LIN {X 0,Y 474.316,Z 460.054,A -85,B 0,C 180,E1 -7102.337,E2 -7102.337} C_VEL
LIN {X 0,Y 474.18,Z 465.59,A -85,B 0,C 180,E1 -7103.233,E2 -7103.233} C_VEL
LIN {X 0,Y 474.066,Z 469.783,A -85,B 0,C 180,E1 -7104.044,E2 -7104.044} C_VEL
LIN {X 0,Y 473.822,Z 474.988,A -85,B 0,C 180,E1 -7105.321,E2 -7105.321} C_VEL
LIN {X 0,Y 473.855,Z 477.663,A -85,B 0,C 180,E1 -7106.173,E2 -7106.173} C_VEL
LIN {X 0,Y 473.746,Z 480.593,A -85,B 0,C 180,E1 -7107.449,E2 -7107.449} C_VEL
LIN {X 0,Y 473.697,Z 481.876,A -85,B 0,C 180,E1 -7108.3,E2 -7108.3} C_VEL
LIN {X 0,Y 473.685,Z 482.688,A -85,B 0,C 180,E1 -7109.15,E2 -7109.15} C_VEL
LIN {X 0,Y 473.668,Z 482.997,A -85,B 0,C 180,E1 -7110,E2 -7110} C_VEL
LIN {X 0,Y 473.686,Z 482.723,A -85,B 0,C 180,E1 -7110.85,E2 -7110.85} C_VEL
LIN {X 0,Y 473.695,Z 481.979,A -85,B 0,C 180,E1 -7111.7,E2 -7111.7} C_VEL
LIN {X 0,Y 473.728,Z 480.766,A -85,B 0,C 180,E1 -7112.551,E2 -7112.551} C_VEL
LIN {X 0,Y 473.852,Z 477.91,A -85,B 0,C 180,E1 -7113.827,E2 -7113.827} C_VEL
LIN {X 0,Y 473.817,Z 475.311,A -85,B 0,C 180,E1 -7114.679,E2 -7114.679} C_VEL
LIN {X 0,Y 474.052,Z 470.192,A -85,B 0,C 180,E1 -7115.957,E2 -7115.957} C_VEL
LIN {X 0,Y 474.188,Z 464.687,A -85,B 0,C 180,E1 -7117.023,E2 -7117.023} C_VEL
LIN {X 0,Y 474.404,Z 457.777,A -85,B 0,C 180,E1 -7118.09,E2 -7118.09} C_VEL
LIN {X 0,Y 474.692,Z 449.845,A -85,B 0,C 180,E1 -7119.05,E2 -7119.05} C_VEL
LIN {X 0,Y 474.987,Z 442.281,A -85,B 0,C 180,E1 -7119.797,E2 -7119.797} C_VEL
LIN {X 0,Y 475.274,Z 434.358,A -85,B 0,C 180,E1 -7120.436,E2 -7120.436} C_VEL
LIN {X 0,Y 475.551,Z 426.183,A -85,B 0,C 180,E1 -7120.969,E2 -7120.969} C_VEL
LIN {X 0,Y 475.774,Z 417.91,A -85,B 0,C 180,E1 -7121.395,E2 -7121.395} C_VEL
LIN {X 0,Y 475.954,Z 408.99,A -85,B 0,C 180,E1 -7121.741,E2 -7121.741} C_VEL
LIN {X 0,Y 476.163,Z 399.664,A -85,B 0,C 180,E1 -7121.987,E2 -7121.987} C_VEL
LIN {X 0,Y 476.373,Z 336.635,A -85,B 0,C 180,E1 -7122.957,E2 -7122.957} C_VEL
LIN {X 0,Y 474.583,Z 324.02,A -85,B 0,C 180,E1 -7123.223,E2 -7123.223} C_VEL
LIN {X 0,Y 474.544,Z 323.281,A -85,B 0,C 180,E1 -7123.314,E2 -7123.314} C_VEL
LIN {X 0,Y 474.924,Z 309.716,A -85,B 0,C 180,E1 -7126.329,E2 -7126.329} C_VEL
LIN {X 0,Y 475.429,Z 296.05,A -85,B 0,C 180,E1 -7129.426,E2 -7129.426} C_VEL
LIN {X 0,Y 475.34,Z 290.192,A -85,B 0,C 180,E1 -7130.783,E2 -7130.783} C_VEL
LIN {X 0,Y 474.664,Z 286.26,A -85,B 0,C 180,E1 -7131.782,E2 -7131.782} C_VEL
LIN {X 0,Y 474.625,Z 286.175,A -85,B 0,C 180,E1 -7134.494,E2 -7134.494} C_VEL
LIN {X 0,Y 474.598,Z 286.18,A -85,B 0,C 180,E1 -7137.326,E2 -7137.326} C_VEL
LIN {X 0,Y 474.594,Z 286.176,A -85,B 0,C 180,E1 -7140.23,E2 -7140.23} C_VEL
LIN {X 0,Y 474.612,Z 286.178,A -85,B 0,C 180,E1 -7143.222,E2 -7143.222} C_VEL
LIN {X 0,Y 474.58,Z 286.177,A -85,B 0,C 180,E1 -7146.323,E2 -7146.323} C_VEL
LIN {X 0,Y 474.618,Z 286.177,A -85,B 0,C 180,E1 -7149.547,E2 -7149.547} C_VEL
LIN {X 0,Y 474.571,Z 286.178,A -85,B 0,C 180,E1 -7152.229,E2 -7152.229} C_VEL
LIN {X 0,Y 474.61,Z 286.18,A -85,B 0,C 180,E1 -7155.297,E2 -7155.297} C_VEL
LIN {X 0,Y 474.585,Z 286.177,A -85,B 0,C 180,E1 -7158.211,E2 -7158.211} C_VEL
LIN {X 0,Y 474.601,Z 286.176,A -85,B 0,C 180,E1 -7161.541,E2 -7161.541} C_VEL
LIN {X 0,Y 474.611,Z 286.179,A -85,B 0,C 180,E1 -7164.724,E2 -7164.724} C_VEL
LIN {X 0,Y 474.617,Z 286.173,A -85,B 0,C 180,E1 -7167.786,E2 -7167.786} C_VEL
LIN {X 0,Y 474.589,Z 286.182,A -85,B 0,C 180,E1 -7170.89,E2 -7170.89} C_VEL
LIN {X 0,Y 474.58,Z 286.177,A -85,B 0,C 180,E1 -7173.623,E2 -7173.623} C_VEL
LIN {X 0,Y 474.624,Z 286.18,A -85,B 0,C 180,E1 -7176.642,E2 -7176.642} C_VEL
LIN {X 0,Y 474.631,Z 286.173,A -85,B 0,C 180,E1 -7180.088,E2 -7180.088} C_VEL
LIN {X 0,Y 474.578,Z 286.181,A -85,B 0,C 180,E1 -7182.772,E2 -7182.772} C_VEL
LIN {X 0,Y 474.621,Z 286.172,A -85,B 0,C 180,E1 -7185.42,E2 -7185.42} C_VEL
LIN {X 0,Y 474.693,Z 286.167,A -85,B 0,C 180,E1 -7188.037,E2 -7188.037} C_VEL
LIN {X 0,Y 474.696,Z 286.163,A -85,B 0,C 180,E1 -7191.486,E2 -7191.486} C_VEL
LIN {X 0,Y 474.728,Z 286.165,A -85,B 0,C 180,E1 -7194.052,E2 -7194.052} C_VEL
LIN {X 0,Y 474.86,Z 286.143,A -85,B 0,C 180,E1 -7197.455,E2 -7197.455} C_VEL
LIN {X 0,Y 474.868,Z 286.149,A -85,B 0,C 180,E1 -7200,E2 -7200} C_VEL
LIN {X 0,Y 474.859,Z 286.144,A -85,B 0,C 180,E1 -7202.545,E2 -7202.545} C_VEL
LIN {X 0,Y 474.726,Z 286.166,A -85,B 0,C 180,E1 -7205.948,E2 -7205.948} C_VEL
LIN {X 0,Y 474.652,Z 286.169,A -85,B 0,C 180,E1 -7208.515,E2 -7208.515} C_VEL
LIN {X 0,Y 474.681,Z 286.169,A -85,B 0,C 180,E1 -7211.963,E2 -7211.963} C_VEL
LIN {X 0,Y 474.676,Z 286.171,A -85,B 0,C 180,E1 -7215.456,E2 -7215.456} C_VEL
LIN {X 0,Y 474.646,Z 286.171,A -85,B 0,C 180,E1 -7219.011,E2 -7219.011} C_VEL
LIN {X 0,Y 474.569,Z 286.183,A -85,B 0,C 180,E1 -7221.73,E2 -7221.73} C_VEL
LIN {X 0,Y 474.614,Z 286.173,A -85,B 0,C 180,E1 -7224.495,E2 -7224.495} C_VEL
LIN {X 0,Y 474.588,Z 286.185,A -85,B 0,C 180,E1 -7227.327,E2 -7227.327} C_VEL
LIN {X 0,Y 474.584,Z 286.177,A -85,B 0,C 180,E1 -7230.232,E2 -7230.232} C_VEL
LIN {X 0,Y 474.605,Z 286.182,A -85,B 0,C 180,E1 -7233.223,E2 -7233.223} C_VEL
LIN {X 0,Y 474.573,Z 286.178,A -85,B 0,C 180,E1 -7236.325,E2 -7236.325} C_VEL
LIN {X 0,Y 474.613,Z 286.175,A -85,B 0,C 180,E1 -7239.549,E2 -7239.549} C_VEL
LIN {X 0,Y 474.568,Z 286.179,A -85,B 0,C 180,E1 -7242.231,E2 -7242.231} C_VEL
LIN {X 0,Y 474.609,Z 286.176,A -85,B 0,C 180,E1 -7245.299,E2 -7245.299} C_VEL
LIN {X 0,Y 474.585,Z 286.178,A -85,B 0,C 180,E1 -7248.212,E2 -7248.212} C_VEL
LIN {X 0,Y 474.612,Z 286.177,A -85,B 0,C 180,E1 -7250.452,E2 -7250.452} C_VEL
LIN {X 0,Y 474.576,Z 286.178,A -85,B 0,C 180,E1 -7253.676,E2 -7253.676} C_VEL
LIN {X 0,Y 474.61,Z 286.179,A -85,B 0,C 180,E1 -7256.778,E2 -7256.778} C_VEL
LIN {X 0,Y 474.59,Z 286.176,A -85,B 0,C 180,E1 -7259.77,E2 -7259.77} C_VEL
LIN {X 0,Y 474.598,Z 286.18,A -85,B 0,C 180,E1 -7262.685,E2 -7262.685} C_VEL
LIN {X 0,Y 474.623,Z 286.175,A -85,B 0,C 180,E1 -7265.506,E2 -7265.506} C_VEL
LIN {X 0,Y 474.712,Z 286.437,A -85,B 0,C 180,E1 -7268.352,E2 -7268.352} C_VEL
LIN {X 0,Y 475.443,Z 291.952,A -85,B 0,C 180,E1 -7269.674,E2 -7269.674} C_VEL
LIN {X 0,Y 475.206,Z 301.711,A -85,B 0,C 180,E1 -7271.906,E2 -7271.906} C_VEL
LIN {X 0,Y 474.769,Z 315.374,A -85,B 0,C 180,E1 -7274.987,E2 -7274.987} C_VEL
LIN {X 0,Y 474.578,Z 323.788,A -85,B 0,C 180,E1 -7276.807,E2 -7276.807} C_VEL
LIN {X 0,Y 475.466,Z 329.742,A -85,B 0,C 180,E1 -7276.958,E2 -7276.958} C_VEL
LIN {X 0,Y 476.52,Z 339.123,A -85,B 0,C 180,E1 -7277.13,E2 -7277.13} C_VEL
LIN {X 0,Y 476.13,Z 399.536,A -85,B 0,C 180,E1 -7278.055,E2 -7278.055} C_VEL
LIN {X 0,Y 475.958,Z 408.436,A -85,B 0,C 180,E1 -7278.286,E2 -7278.286} C_VEL
LIN {X 0,Y 475.82,Z 418.11,A -85,B 0,C 180,E1 -7278.66,E2 -7278.66} C_VEL
LIN {X 0,Y 475.509,Z 427.274,A -85,B 0,C 180,E1 -7279.138,E2 -7279.138} C_VEL
LIN {X 0,Y 475.138,Z 438.077,A -85,B 0,C 180,E1 -7279.884,E2 -7279.884} C_VEL
LIN {X 0,Y 474.823,Z 447.376,A -85,B 0,C 180,E1 -7280.737,E2 -7280.737} C_VEL
LIN {X 0,Y 474.522,Z 454.038,A -85,B 0,C 180,E1 -7281.483,E2 -7281.483} C_VEL
LIN {X 0,Y 474.314,Z 460.361,A -85,B 0,C 180,E1 -7282.337,E2 -7282.337} C_VEL
LIN {X 0,Y 474.177,Z 465.856,A -85,B 0,C 180,E1 -7283.235,E2 -7283.235} C_VEL
LIN {X 0,Y 474.067,Z 469.991,A -85,B 0,C 180,E1 -7284.044,E2 -7284.044} C_VEL
LIN {X 0,Y 473.818,Z 475.151,A -85,B 0,C 180,E1 -7285.321,E2 -7285.321} C_VEL
LIN {X 0,Y 473.832,Z 478.939,A -85,B 0,C 180,E1 -7286.599,E2 -7286.599} C_VEL
LIN {X 0,Y 473.745,Z 480.681,A -85,B 0,C 180,E1 -7287.449,E2 -7287.449} C_VEL
LIN {X 0,Y 473.697,Z 481.928,A -85,B 0,C 180,E1 -7288.3,E2 -7288.3} C_VEL
LIN {X 0,Y 473.685,Z 482.706,A -85,B 0,C 180,E1 -7289.15,E2 -7289.15} C_VEL
LIN {X 0,Y 473.666,Z 483,A -85,B 0,C 180,E1 -7290,E2 -7290} C_VEL
LIN {X 0,Y 473.685,Z 482.705,A -85,B 0,C 180,E1 -7290.85,E2 -7290.85} C_VEL
LIN {X 0,Y 473.697,Z 481.927,A -85,B 0,C 180,E1 -7291.7,E2 -7291.7} C_VEL
LIN {X 0,Y 473.745,Z 480.678,A -85,B 0,C 180,E1 -7292.551,E2 -7292.551} C_VEL
LIN {X 0,Y 473.853,Z 477.785,A -85,B 0,C 180,E1 -7293.827,E2 -7293.827} C_VEL
LIN {X 0,Y 473.818,Z 475.148,A -85,B 0,C 180,E1 -7294.679,E2 -7294.679} C_VEL
LIN {X 0,Y 474.066,Z 469.984,A -85,B 0,C 180,E1 -7295.956,E2 -7295.956} C_VEL
LIN {X 0,Y 474.226,Z 463.18,A -85,B 0,C 180,E1 -7297.237,E2 -7297.237} C_VEL
LIN {X 0,Y 474.452,Z 455.736,A -85,B 0,C 180,E1 -7298.304,E2 -7298.304} C_VEL
LIN {X 0,Y 474.762,Z 448.394,A -85,B 0,C 180,E1 -7299.156,E2 -7299.156} C_VEL
LIN {X 0,Y 475.044,Z 440.529,A -85,B 0,C 180,E1 -7299.903,E2 -7299.903} C_VEL
LIN {X 0,Y 475.369,Z 432.217,A -85,B 0,C 180,E1 -7300.542,E2 -7300.542} C_VEL
LIN {X 0,Y 475.696,Z 421.603,A -85,B 0,C 180,E1 -7301.181,E2 -7301.181} C_VEL
LIN {X 0,Y 475.937,Z 410.065,A -85,B 0,C 180,E1 -7301.661,E2 -7301.661} C_VEL
LIN {X 0,Y 476.13,Z 400.422,A -85,B 0,C 180,E1 -7301.926,E2 -7301.926} C_VEL
LIN {X 0,Y 476.344,Z 336.118,A -85,B 0,C 180,E1 -7302.92,E2 -7302.92} C_VEL
LIN {X 0,Y 474.557,Z 324.126,A -85,B 0,C 180,E1 -7303.168,E2 -7303.168} C_VEL
LIN {X 0,Y 474.553,Z 322.198,A -85,B 0,C 180,E1 -7303.489,E2 -7303.489} C_VEL
LIN {X 0,Y 474.923,Z 309.51,A -85,B 0,C 180,E1 -7306.329,E2 -7306.329} C_VEL
LIN {X 0,Y 475.428,Z 295.845,A -85,B 0,C 180,E1 -7309.426,E2 -7309.426} C_VEL
LIN {X 0,Y 475.31,Z 289.988,A -85,B 0,C 180,E1 -7310.785,E2 -7310.785} C_VEL
LIN {X 0,Y 474.664,Z 286.269,A -85,B 0,C 180,E1 -7311.725,E2 -7311.725} C_VEL
LIN {X 0,Y 474.623,Z 286.175,A -85,B 0,C 180,E1 -7314.494,E2 -7314.494} C_VEL
LIN {X 0,Y 474.596,Z 286.18,A -85,B 0,C 180,E1 -7317.326,E2 -7317.326} C_VEL
LIN {X 0,Y 474.59,Z 286.176,A -85,B 0,C 180,E1 -7320.23,E2 -7320.23} C_VEL
LIN {X 0,Y 474.61,Z 286.179,A -85,B 0,C 180,E1 -7323.222,E2 -7323.222} C_VEL
LIN {X 0,Y 474.576,Z 286.178,A -85,B 0,C 180,E1 -7326.324,E2 -7326.324} C_VEL
LIN {X 0,Y 474.616,Z 286.177,A -85,B 0,C 180,E1 -7329.548,E2 -7329.548} C_VEL
LIN {X 0,Y 474.57,Z 286.178,A -85,B 0,C 180,E1 -7332.229,E2 -7332.229} C_VEL
LIN {X 0,Y 474.609,Z 286.179,A -85,B 0,C 180,E1 -7335.297,E2 -7335.297} C_VEL
LIN {X 0,Y 474.584,Z 286.177,A -85,B 0,C 180,E1 -7338.211,E2 -7338.211} C_VEL
LIN {X 0,Y 474.599,Z 286.176,A -85,B 0,C 180,E1 -7341.542,E2 -7341.542} C_VEL
LIN {X 0,Y 474.608,Z 286.18,A -85,B 0,C 180,E1 -7344.724,E2 -7344.724} C_VEL
LIN {X 0,Y 474.616,Z 286.173,A -85,B 0,C 180,E1 -7347.786,E2 -7347.786} C_VEL
LIN {X 0,Y 474.588,Z 286.182,A -85,B 0,C 180,E1 -7350.89,E2 -7350.89} C_VEL
LIN {X 0,Y 474.58,Z 286.177,A -85,B 0,C 180,E1 -7353.624,E2 -7353.624} C_VEL
LIN {X 0,Y 474.623,Z 286.179,A -85,B 0,C 180,E1 -7356.642,E2 -7356.642} C_VEL
LIN {X 0,Y 474.631,Z 286.174,A -85,B 0,C 180,E1 -7360.089,E2 -7360.089} C_VEL
LIN {X 0,Y 474.577,Z 286.181,A -85,B 0,C 180,E1 -7362.772,E2 -7362.772} C_VEL
LIN {X 0,Y 474.62,Z 286.172,A -85,B 0,C 180,E1 -7365.42,E2 -7365.42} C_VEL
LIN {X 0,Y 474.693,Z 286.167,A -85,B 0,C 180,E1 -7368.037,E2 -7368.037} C_VEL
LIN {X 0,Y 474.684,Z 286.165,A -85,B 0,C 180,E1 -7371.486,E2 -7371.486} C_VEL
LIN {X 0,Y 474.727,Z 286.165,A -85,B 0,C 180,E1 -7374.052,E2 -7374.052} C_VEL
LIN {X 0,Y 474.86,Z 286.143,A -85,B 0,C 180,E1 -7377.455,E2 -7377.455} C_VEL
LIN {X 0,Y 474.868,Z 286.149,A -85,B 0,C 180,E1 -7380,E2 -7380} C_VEL
LIN {X 0,Y 474.859,Z 286.144,A -85,B 0,C 180,E1 -7382.545,E2 -7382.545} C_VEL
LIN {X 0,Y 474.727,Z 286.166,A -85,B 0,C 180,E1 -7385.948,E2 -7385.948} C_VEL
LIN {X 0,Y 474.649,Z 286.169,A -85,B 0,C 180,E1 -7388.515,E2 -7388.515} C_VEL
LIN {X 0,Y 474.681,Z 286.17,A -85,B 0,C 180,E1 -7391.963,E2 -7391.963} C_VEL
LIN {X 0,Y 474.677,Z 286.171,A -85,B 0,C 180,E1 -7395.457,E2 -7395.457} C_VEL
LIN {X 0,Y 474.647,Z 286.171,A -85,B 0,C 180,E1 -7399.011,E2 -7399.011} C_VEL
LIN {X 0,Y 474.57,Z 286.183,A -85,B 0,C 180,E1 -7401.73,E2 -7401.73} C_VEL
LIN {X 0,Y 474.614,Z 286.173,A -85,B 0,C 180,E1 -7404.495,E2 -7404.495} C_VEL
LIN {X 0,Y 474.588,Z 286.184,A -85,B 0,C 180,E1 -7407.327,E2 -7407.327} C_VEL
LIN {X 0,Y 474.571,Z 286.178,A -85,B 0,C 180,E1 -7410.233,E2 -7410.233} C_VEL
LIN {X 0,Y 474.605,Z 286.182,A -85,B 0,C 180,E1 -7413.223,E2 -7413.223} C_VEL
LIN {X 0,Y 474.573,Z 286.178,A -85,B 0,C 180,E1 -7416.325,E2 -7416.325} C_VEL
LIN {X 0,Y 474.594,Z 286.177,A -85,B 0,C 180,E1 -7419.644,E2 -7419.644} C_VEL
LIN {X 0,Y 474.562,Z 286.187,A -85,B 0,C 180,E1 -7422.94,E2 -7422.94} C_VEL
LIN {X 0,Y 474.596,Z 286.175,A -85,B 0,C 180,E1 -7425.895,E2 -7425.895} C_VEL
LIN {X 0,Y 474.586,Z 286.178,A -85,B 0,C 180,E1 -7429.34,E2 -7429.34} C_VEL
LIN {X 0,Y 474.59,Z 286.176,A -85,B 0,C 180,E1 -7431.707,E2 -7431.707} C_VEL
LIN {X 0,Y 474.613,Z 286.181,A -85,B 0,C 180,E1 -7434.726,E2 -7434.726} C_VEL
LIN {X 0,Y 474.622,Z 286.172,A -85,B 0,C 180,E1 -7437.788,E2 -7437.788} C_VEL
LIN {X 0,Y 474.575,Z 286.181,A -85,B 0,C 180,E1 -7440.896,E2 -7440.896} C_VEL
LIN {X 0,Y 474.588,Z 286.176,A -85,B 0,C 180,E1 -7443.625,E2 -7443.625} C_VEL
LIN {X 0,Y 474.596,Z 286.164,A -85,B 0,C 180,E1 -7446.653,E2 -7446.653} C_VEL
LIN {X 0,Y 474.668,Z 286.308,A -85,B 0,C 180,E1 -7448.352,E2 -7448.352} C_VEL
LIN {X 0,Y 475.4,Z 291.748,A -85,B 0,C 180,E1 -7449.672,E2 -7449.672} C_VEL
LIN {X 0,Y 475.335,Z 298.788,A -85,B 0,C 180,E1 -7451.29,E2 -7451.29} C_VEL
LIN {X 0,Y 474.577,Z 301.622,A -85,B 0,C 180,E1 -7451.908,E2 -7451.908} C_VEL
LIN {X 0,Y 468.5,Z 311.263,A -85,B 0,C 180,E1 -7453.888,E2 -7453.888} C_VEL
LIN {X 0,Y 467.768,Z 314.124,A -85,B 0,C 180,E1 -7454.517,E2 -7454.517} C_VEL
LIN {X 0,Y 467.515,Z 323.768,A -85,B 0,C 180,E1 -7456.648,E2 -7456.648} C_VEL
LIN {X 0,Y 468.37,Z 329.459,A -85,B 0,C 180,E1 -7456.799,E2 -7456.799} C_VEL
LIN {X 0,Y 469.555,Z 338.791,A -85,B 0,C 180,E1 -7456.977,E2 -7456.977} C_VEL
LIN {X 0,Y 469.267,Z 399.579,A -85,B 0,C 180,E1 -7457.925,E2 -7457.925} C_VEL
LIN {X 0,Y 469.039,Z 408.693,A -85,B 0,C 180,E1 -7458.165,E2 -7458.165} C_VEL
LIN {X 0,Y 468.863,Z 417.089,A -85,B 0,C 180,E1 -7458.49,E2 -7458.49} C_VEL
LIN {X 0,Y 468.573,Z 424.61,A -85,B 0,C 180,E1 -7458.866,E2 -7458.866} C_VEL
LIN {X 0,Y 468.361,Z 433.096,A -85,B 0,C 180,E1 -7459.408,E2 -7459.408} C_VEL
LIN {X 0,Y 468.059,Z 441.249,A -85,B 0,C 180,E1 -7460.057,E2 -7460.057} C_VEL
LIN {X 0,Y 467.704,Z 448.991,A -85,B 0,C 180,E1 -7460.813,E2 -7460.813} C_VEL
LIN {X 0,Y 467.374,Z 457.084,A -85,B 0,C 180,E1 -7461.787,E2 -7461.787} C_VEL
LIN {X 0,Y 467.165,Z 464.185,A -85,B 0,C 180,E1 -7462.871,E2 -7462.871} C_VEL
LIN {X 0,Y 466.99,Z 469.785,A -85,B 0,C 180,E1 -7463.953,E2 -7463.953} C_VEL
LIN {X 0,Y 466.746,Z 474.989,A -85,B 0,C 180,E1 -7465.25,E2 -7465.25} C_VEL
LIN {X 0,Y 466.765,Z 477.665,A -85,B 0,C 180,E1 -7466.115,E2 -7466.115} C_VEL
LIN {X 0,Y 466.668,Z 480.593,A -85,B 0,C 180,E1 -7467.411,E2 -7467.411} C_VEL
LIN {X 0,Y 466.607,Z 481.876,A -85,B 0,C 180,E1 -7468.274,E2 -7468.274} C_VEL
LIN {X 0,Y 466.587,Z 482.688,A -85,B 0,C 180,E1 -7469.137,E2 -7469.137} C_VEL
LIN {X 0,Y 466.568,Z 482.997,A -85,B 0,C 180,E1 -7470,E2 -7470} C_VEL
LIN {X 0,Y 466.588,Z 482.722,A -85,B 0,C 180,E1 -7470.863,E2 -7470.863} C_VEL
LIN {X 0,Y 466.604,Z 481.979,A -85,B 0,C 180,E1 -7471.726,E2 -7471.726} C_VEL
LIN {X 0,Y 466.652,Z 480.765,A -85,B 0,C 180,E1 -7472.59,E2 -7472.59} C_VEL
LIN {X 0,Y 466.762,Z 477.908,A -85,B 0,C 180,E1 -7473.885,E2 -7473.885} C_VEL
LIN {X 0,Y 466.741,Z 475.31,A -85,B 0,C 180,E1 -7474.75,E2 -7474.75} C_VEL
LIN {X 0,Y 466.977,Z 470.19,A -85,B 0,C 180,E1 -7476.047,E2 -7476.047} C_VEL
LIN {X 0,Y 467.132,Z 464.684,A -85,B 0,C 180,E1 -7477.13,E2 -7477.13} C_VEL
LIN {X 0,Y 467.366,Z 457.774,A -85,B 0,C 180,E1 -7478.213,E2 -7478.213} C_VEL
LIN {X 0,Y 467.699,Z 449.841,A -85,B 0,C 180,E1 -7479.187,E2 -7479.187} C_VEL
LIN {X 0,Y 468.003,Z 442.276,A -85,B 0,C 180,E1 -7479.944,E2 -7479.944} C_VEL
LIN {X 0,Y 468.3,Z 434.352,A -85,B 0,C 180,E1 -7480.593,E2 -7480.593} C_VEL
LIN {X 0,Y 468.564,Z 426.175,A -85,B 0,C 180,E1 -7481.134,E2 -7481.134} C_VEL
LIN {X 0,Y 468.828,Z 417.899,A -85,B 0,C 180,E1 -7481.566,E2 -7481.566} C_VEL
LIN {X 0,Y 469.005,Z 408.976,A -85,B 0,C 180,E1 -7481.918,E2 -7481.918} C_VEL
LIN {X 0,Y 469.227,Z 399.791,A -85,B 0,C 180,E1 -7482.164,E2 -7482.164} C_VEL
LIN {X 0,Y 469.436,Z 337.006,A -85,B 0,C 180,E1 -7483.146,E2 -7483.146} C_VEL
LIN {X 0,Y 467.546,Z 324.012,A -85,B 0,C 180,E1 -7483.426,E2 -7483.426} C_VEL
LIN {X 0,Y 467.505,Z 323.278,A -85,B 0,C 180,E1 -7483.518,E2 -7483.518} C_VEL
LIN {X 0,Y 467.925,Z 309.714,A -85,B 0,C 180,E1 -7486.581,E2 -7486.581} C_VEL
LIN {X 0,Y 468.395,Z 298,A -85,B 0,C 180,E1 -7489.274,E2 -7489.274} C_VEL
LIN {X 0,Y 468.412,Z 292.143,A -85,B 0,C 180,E1 -7490.645,E2 -7490.645} C_VEL
LIN {X 0,Y 467.638,Z 287.13,A -85,B 0,C 180,E1 -7491.921,E2 -7491.921} C_VEL
LIN {X 0,Y 467.558,Z 287.055,A -85,B 0,C 180,E1 -7494.889,E2 -7494.889} C_VEL
LIN {X 0,Y 467.544,Z 287.059,A -85,B 0,C 180,E1 -7497.773,E2 -7497.773} C_VEL
LIN {X 0,Y 467.563,Z 287.054,A -85,B 0,C 180,E1 -7501.043,E2 -7501.043} C_VEL
LIN {X 0,Y 467.573,Z 287.05,A -85,B 0,C 180,E1 -7504.239,E2 -7504.239} C_VEL
LIN {X 0,Y 467.538,Z 287.06,A -85,B 0,C 180,E1 -7507.184,E2 -7507.184} C_VEL
LIN {X 0,Y 467.553,Z 287.053,A -85,B 0,C 180,E1 -7510.266,E2 -7510.266} C_VEL
LIN {X 0,Y 467.539,Z 287.056,A -85,B 0,C 180,E1 -7513.745,E2 -7513.745} C_VEL
LIN {X 0,Y 467.538,Z 287.055,A -85,B 0,C 180,E1 -7516.253,E2 -7516.253} C_VEL
LIN {X 0,Y 467.55,Z 287.054,A -85,B 0,C 180,E1 -7519.732,E2 -7519.732} C_VEL
LIN {X 0,Y 467.535,Z 287.061,A -85,B 0,C 180,E1 -7522.814,E2 -7522.814} C_VEL
LIN {X 0,Y 467.568,Z 287.051,A -85,B 0,C 180,E1 -7525.76,E2 -7525.76} C_VEL
LIN {X 0,Y 467.538,Z 287.06,A -85,B 0,C 180,E1 -7528.959,E2 -7528.959} C_VEL
LIN {X 0,Y 467.536,Z 287.057,A -85,B 0,C 180,E1 -7532.225,E2 -7532.225} C_VEL
LIN {X 0,Y 467.549,Z 287.055,A -85,B 0,C 180,E1 -7535.109,E2 -7535.109} C_VEL
LIN {X 0,Y 467.516,Z 287.058,A -85,B 0,C 180,E1 -7537.925,E2 -7537.925} C_VEL
LIN {X 0,Y 467.606,Z 287.052,A -85,B 0,C 180,E1 -7540.691,E2 -7540.691} C_VEL
LIN {X 0,Y 467.601,Z 287.053,A -85,B 0,C 180,E1 -7544.304,E2 -7544.304} C_VEL
LIN {X 0,Y 467.645,Z 287.043,A -85,B 0,C 180,E1 -7547.854,E2 -7547.854} C_VEL
LIN {X 0,Y 467.655,Z 287.04,A -85,B 0,C 180,E1 -7551.357,E2 -7551.357} C_VEL
LIN {X 0,Y 467.693,Z 287.04,A -85,B 0,C 180,E1 -7553.962,E2 -7553.962} C_VEL
LIN {X 0,Y 467.801,Z 287.023,A -85,B 0,C 180,E1 -7557.417,E2 -7557.417} C_VEL
LIN {X 0,Y 467.837,Z 287.025,A -85,B 0,C 180,E1 -7560,E2 -7560} C_VEL
LIN {X 0,Y 467.8,Z 287.023,A -85,B 0,C 180,E1 -7562.583,E2 -7562.583} C_VEL
LIN {X 0,Y 467.691,Z 287.041,A -85,B 0,C 180,E1 -7566.038,E2 -7566.038} C_VEL
LIN {X 0,Y 467.621,Z 287.044,A -85,B 0,C 180,E1 -7568.644,E2 -7568.644} C_VEL
LIN {X 0,Y 467.636,Z 287.045,A -85,B 0,C 180,E1 -7572.146,E2 -7572.146} C_VEL
LIN {X 0,Y 467.601,Z 287.054,A -85,B 0,C 180,E1 -7575.696,E2 -7575.696} C_VEL
LIN {X 0,Y 467.604,Z 287.051,A -85,B 0,C 180,E1 -7579.308,E2 -7579.308} C_VEL
LIN {X 0,Y 467.513,Z 287.059,A -85,B 0,C 180,E1 -7582.075,E2 -7582.075} C_VEL
LIN {X 0,Y 467.548,Z 287.055,A -85,B 0,C 180,E1 -7584.89,E2 -7584.89} C_VEL
LIN {X 0,Y 467.534,Z 287.057,A -85,B 0,C 180,E1 -7587.774,E2 -7587.774} C_VEL
LIN {X 0,Y 467.537,Z 287.06,A -85,B 0,C 180,E1 -7591.041,E2 -7591.041} C_VEL
LIN {X 0,Y 467.567,Z 287.051,A -85,B 0,C 180,E1 -7594.24,E2 -7594.24} C_VEL
LIN {X 0,Y 467.533,Z 287.062,A -85,B 0,C 180,E1 -7597.186,E2 -7597.186} C_VEL
LIN {X 0,Y 467.549,Z 287.054,A -85,B 0,C 180,E1 -7600.267,E2 -7600.267} C_VEL
LIN {X 0,Y 467.537,Z 287.055,A -85,B 0,C 180,E1 -7603.746,E2 -7603.746} C_VEL
LIN {X 0,Y 467.538,Z 287.056,A -85,B 0,C 180,E1 -7606.255,E2 -7606.255} C_VEL
LIN {X 0,Y 467.55,Z 287.053,A -85,B 0,C 180,E1 -7609.734,E2 -7609.734} C_VEL
LIN {X 0,Y 467.532,Z 287.062,A -85,B 0,C 180,E1 -7612.816,E2 -7612.816} C_VEL
LIN {X 0,Y 467.571,Z 287.05,A -85,B 0,C 180,E1 -7615.761,E2 -7615.761} C_VEL
LIN {X 0,Y 467.543,Z 287.057,A -85,B 0,C 180,E1 -7618.96,E2 -7618.96} C_VEL
LIN {X 0,Y 467.541,Z 287.059,A -85,B 0,C 180,E1 -7622.227,E2 -7622.227} C_VEL
LIN {X 0,Y 467.556,Z 287.056,A -85,B 0,C 180,E1 -7625.111,E2 -7625.111} C_VEL
LIN {X 0,Y 467.642,Z 287.208,A -85,B 0,C 180,E1 -7628.178,E2 -7628.178} C_VEL
LIN {X 0,Y 468.476,Z 293.905,A -85,B 0,C 180,E1 -7629.816,E2 -7629.816} C_VEL
LIN {X 0,Y 468.159,Z 303.664,A -85,B 0,C 180,E1 -7632.077,E2 -7632.077} C_VEL
LIN {X 0,Y 467.657,Z 317.327,A -85,B 0,C 180,E1 -7635.198,E2 -7635.198} C_VEL
LIN {X 0,Y 467.51,Z 323.676,A -85,B 0,C 180,E1 -7636.592,E2 -7636.592} C_VEL
LIN {X 0,Y 468.039,Z 327.4,A -85,B 0,C 180,E1 -7636.711,E2 -7636.711} C_VEL
LIN {X 0,Y 469.62,Z 339.462,A -85,B 0,C 180,E1 -7636.942,E2 -7636.942} C_VEL
LIN {X 0,Y 469.194,Z 399.594,A -85,B 0,C 180,E1 -7637.876,E2 -7637.876} C_VEL
LIN {X 0,Y 469,Z 409.275,A -85,B 0,C 180,E1 -7638.137,E2 -7638.137} C_VEL
LIN {X 0,Y 468.853,Z 419.325,A -85,B 0,C 180,E1 -7638.544,E2 -7638.544} C_VEL
LIN {X 0,Y 468.43,Z 430.734,A -85,B 0,C 180,E1 -7639.191,E2 -7639.191} C_VEL
LIN {X 0,Y 468.124,Z 439.312,A -85,B 0,C 180,E1 -7639.84,E2 -7639.84} C_VEL
LIN {X 0,Y 467.807,Z 447.378,A -85,B 0,C 180,E1 -7640.597,E2 -7640.597} C_VEL
LIN {X 0,Y 467.495,Z 454.04,A -85,B 0,C 180,E1 -7641.354,E2 -7641.354} C_VEL
LIN {X 0,Y 467.253,Z 460.362,A -85,B 0,C 180,E1 -7642.22,E2 -7642.22} C_VEL
LIN {X 0,Y 467.116,Z 466.321,A -85,B 0,C 180,E1 -7643.218,E2 -7643.218} C_VEL
LIN {X 0,Y 466.915,Z 471.902,A -85,B 0,C 180,E1 -7644.385,E2 -7644.385} C_VEL
LIN {X 0,Y 466.712,Z 476.623,A -85,B 0,C 180,E1 -7645.682,E2 -7645.682} C_VEL
LIN {X 0,Y 466.734,Z 478.94,A -85,B 0,C 180,E1 -7646.547,E2 -7646.547} C_VEL
LIN {X 0,Y 466.667,Z 480.681,A -85,B 0,C 180,E1 -7647.411,E2 -7647.411} C_VEL
LIN {X 0,Y 466.606,Z 481.929,A -85,B 0,C 180,E1 -7648.274,E2 -7648.274} C_VEL
LIN {X 0,Y 466.587,Z 482.706,A -85,B 0,C 180,E1 -7649.137,E2 -7649.137} C_VEL
LIN {X 0,Y 466.567,Z 483,A -85,B 0,C 180,E1 -7650,E2 -7650} C_VEL
LIN {X 0,Y 466.587,Z 482.705,A -85,B 0,C 180,E1 -7650.863,E2 -7650.863} C_VEL
LIN {X 0,Y 466.606,Z 481.927,A -85,B 0,C 180,E1 -7651.726,E2 -7651.726} C_VEL
LIN {X 0,Y 466.667,Z 480.678,A -85,B 0,C 180,E1 -7652.589,E2 -7652.589} C_VEL
LIN {X 0,Y 466.763,Z 477.784,A -85,B 0,C 180,E1 -7653.885,E2 -7653.885} C_VEL
LIN {X 0,Y 466.742,Z 475.147,A -85,B 0,C 180,E1 -7654.75,E2 -7654.75} C_VEL
LIN {X 0,Y 466.989,Z 469.983,A -85,B 0,C 180,E1 -7656.047,E2 -7656.047} C_VEL
LIN {X 0,Y 467.174,Z 463.178,A -85,B 0,C 180,E1 -7657.346,E2 -7657.346} C_VEL
LIN {X 0,Y 467.427,Z 455.735,A -85,B 0,C 180,E1 -7658.43,E2 -7658.43} C_VEL
LIN {X 0,Y 467.754,Z 448.391,A -85,B 0,C 180,E1 -7659.295,E2 -7659.295} C_VEL
LIN {X 0,Y 468.043,Z 440.526,A -85,B 0,C 180,E1 -7660.053,E2 -7660.053} C_VEL
LIN {X 0,Y 468.401,Z 432.213,A -85,B 0,C 180,E1 -7660.7,E2 -7660.7} C_VEL
LIN {X 0,Y 468.729,Z 421.599,A -85,B 0,C 180,E1 -7661.349,E2 -7661.349} C_VEL
LIN {X 0,Y 469.006,Z 410.058,A -85,B 0,C 180,E1 -7661.835,E2 -7661.835} C_VEL
LIN {X 0,Y 469.193,Z 400.411,A -85,B 0,C 180,E1 -7662.105,E2 -7662.105} C_VEL
LIN {X 0,Y 469.469,Z 337.085,A -85,B 0,C 180,E1 -7663.097,E2 -7663.097} C_VEL
LIN {X 0,Y 467.557,Z 324.429,A -85,B 0,C 180,E1 -7663.359,E2 -7663.359} C_VEL
LIN {X 0,Y 467.507,Z 323.261,A -85,B 0,C 180,E1 -7663.474,E2 -7663.474} C_VEL
LIN {X 0,Y 467.924,Z 309.509,A -85,B 0,C 180,E1 -7666.581,E2 -7666.581} C_VEL
LIN {X 0,Y 468.395,Z 297.796,A -85,B 0,C 180,E1 -7669.274,E2 -7669.274} C_VEL
LIN {X 0,Y 468.388,Z 291.939,A -85,B 0,C 180,E1 -7670.646,E2 -7670.646} C_VEL
LIN {X 0,Y 467.613,Z 287.138,A -85,B 0,C 180,E1 -7671.871,E2 -7671.871} C_VEL
LIN {X 0,Y 467.556,Z 287.056,A -85,B 0,C 180,E1 -7674.889,E2 -7674.889} C_VEL
LIN {X 0,Y 467.542,Z 287.059,A -85,B 0,C 180,E1 -7677.773,E2 -7677.773} C_VEL
LIN {X 0,Y 467.543,Z 287.057,A -85,B 0,C 180,E1 -7681.04,E2 -7681.04} C_VEL
LIN {X 0,Y 467.571,Z 287.05,A -85,B 0,C 180,E1 -7684.239,E2 -7684.239} C_VEL
LIN {X 0,Y 467.536,Z 287.061,A -85,B 0,C 180,E1 -7687.184,E2 -7687.184} C_VEL
LIN {X 0,Y 467.551,Z 287.053,A -85,B 0,C 180,E1 -7690.266,E2 -7690.266} C_VEL
LIN {X 0,Y 467.538,Z 287.056,A -85,B 0,C 180,E1 -7693.745,E2 -7693.745} C_VEL
LIN {X 0,Y 467.537,Z 287.055,A -85,B 0,C 180,E1 -7696.254,E2 -7696.254} C_VEL
LIN {X 0,Y 467.549,Z 287.054,A -85,B 0,C 180,E1 -7699.733,E2 -7699.733} C_VEL
LIN {X 0,Y 467.533,Z 287.062,A -85,B 0,C 180,E1 -7702.814,E2 -7702.814} C_VEL
LIN {X 0,Y 467.567,Z 287.051,A -85,B 0,C 180,E1 -7705.76,E2 -7705.76} C_VEL
LIN {X 0,Y 467.537,Z 287.06,A -85,B 0,C 180,E1 -7708.959,E2 -7708.959} C_VEL
LIN {X 0,Y 467.535,Z 287.057,A -85,B 0,C 180,E1 -7712.226,E2 -7712.226} C_VEL
LIN {X 0,Y 467.549,Z 287.055,A -85,B 0,C 180,E1 -7715.11,E2 -7715.11} C_VEL
LIN {X 0,Y 467.515,Z 287.058,A -85,B 0,C 180,E1 -7717.925,E2 -7717.925} C_VEL
LIN {X 0,Y 467.605,Z 287.051,A -85,B 0,C 180,E1 -7720.692,E2 -7720.692} C_VEL
LIN {X 0,Y 467.601,Z 287.053,A -85,B 0,C 180,E1 -7724.304,E2 -7724.304} C_VEL
LIN {X 0,Y 467.645,Z 287.043,A -85,B 0,C 180,E1 -7727.854,E2 -7727.854} C_VEL
LIN {X 0,Y 467.645,Z 287.041,A -85,B 0,C 180,E1 -7731.357,E2 -7731.357} C_VEL
LIN {X 0,Y 467.692,Z 287.041,A -85,B 0,C 180,E1 -7733.962,E2 -7733.962} C_VEL
LIN {X 0,Y 467.8,Z 287.023,A -85,B 0,C 180,E1 -7737.417,E2 -7737.417} C_VEL
LIN {X 0,Y 467.837,Z 287.025,A -85,B 0,C 180,E1 -7740,E2 -7740} C_VEL
LIN {X 0,Y 467.8,Z 287.023,A -85,B 0,C 180,E1 -7742.583,E2 -7742.583} C_VEL
LIN {X 0,Y 467.691,Z 287.041,A -85,B 0,C 180,E1 -7746.038,E2 -7746.038} C_VEL
LIN {X 0,Y 467.618,Z 287.045,A -85,B 0,C 180,E1 -7748.644,E2 -7748.644} C_VEL
LIN {X 0,Y 467.637,Z 287.045,A -85,B 0,C 180,E1 -7752.146,E2 -7752.146} C_VEL
LIN {X 0,Y 467.602,Z 287.054,A -85,B 0,C 180,E1 -7755.696,E2 -7755.696} C_VEL
LIN {X 0,Y 467.605,Z 287.051,A -85,B 0,C 180,E1 -7759.309,E2 -7759.309} C_VEL
LIN {X 0,Y 467.514,Z 287.059,A -85,B 0,C 180,E1 -7762.075,E2 -7762.075} C_VEL
LIN {X 0,Y 467.548,Z 287.055,A -85,B 0,C 180,E1 -7764.891,E2 -7764.891} C_VEL
LIN {X 0,Y 467.534,Z 287.058,A -85,B 0,C 180,E1 -7767.775,E2 -7767.775} C_VEL
LIN {X 0,Y 467.528,Z 287.061,A -85,B 0,C 180,E1 -7771.039,E2 -7771.039} C_VEL
LIN {X 0,Y 467.568,Z 287.051,A -85,B 0,C 180,E1 -7774.24,E2 -7774.24} C_VEL
LIN {X 0,Y 467.53,Z 287.063,A -85,B 0,C 180,E1 -7777.185,E2 -7777.185} C_VEL
LIN {X 0,Y 467.549,Z 287.053,A -85,B 0,C 180,E1 -7780.268,E2 -7780.268} C_VEL
LIN {X 0,Y 467.538,Z 287.055,A -85,B 0,C 180,E1 -7783.747,E2 -7783.747} C_VEL
LIN {X 0,Y 467.539,Z 287.055,A -85,B 0,C 180,E1 -7786.255,E2 -7786.255} C_VEL
LIN {X 0,Y 467.551,Z 287.053,A -85,B 0,C 180,E1 -7789.734,E2 -7789.734} C_VEL
LIN {X 0,Y 467.533,Z 287.062,A -85,B 0,C 180,E1 -7792.816,E2 -7792.816} C_VEL
LIN {X 0,Y 467.572,Z 287.05,A -85,B 0,C 180,E1 -7795.761,E2 -7795.761} C_VEL
LIN {X 0,Y 467.532,Z 287.058,A -85,B 0,C 180,E1 -7798.963,E2 -7798.963} C_VEL
LIN {X 0,Y 467.538,Z 287.059,A -85,B 0,C 180,E1 -7802.226,E2 -7802.226} C_VEL
LIN {X 0,Y 467.557,Z 287.056,A -85,B 0,C 180,E1 -7805.111,E2 -7805.111} C_VEL
LIN {X 0,Y 467.622,Z 287.234,A -85,B 0,C 180,E1 -7808.235,E2 -7808.235} C_VEL
LIN {X 0,Y 468.442,Z 293.701,A -85,B 0,C 180,E1 -7809.815,E2 -7809.815} C_VEL
LIN {X 0,Y 468.162,Z 303.459,A -85,B 0,C 180,E1 -7812.077,E2 -7812.077} C_VEL
LIN {X 0,Y 467.768,Z 314.124,A -85,B 0,C 180,E1 -7814.517,E2 -7814.517} C_VEL
LIN {X 0,Y 467.026,Z 315.224,A -85,B 0,C 180,E1 -7814.744,E2 -7814.744} C_VEL
LIN {X 0,Y 461.119,Z 318.714,A -85,B 0,C 180,E1 -7815.352,E2 -7815.352} C_VEL
LIN {X 0,Y 460.563,Z 319.641,A -85,B 0,C 180,E1 -7815.548,E2 -7815.548} C_VEL
LIN {X 0,Y 460.482,Z 323.771,A -85,B 0,C 180,E1 -7816.44,E2 -7816.44} C_VEL
LIN {X 0,Y 461.347,Z 329.228,A -85,B 0,C 180,E1 -7816.59,E2 -7816.59} C_VEL
LIN {X 0,Y 462.639,Z 338.819,A -85,B 0,C 180,E1 -7816.779,E2 -7816.779} C_VEL
LIN {X 0,Y 462.341,Z 399.6,A -85,B 0,C 180,E1 -7817.741,E2 -7817.741} C_VEL
LIN {X 0,Y 462.111,Z 408.707,A -85,B 0,C 180,E1 -7817.985,E2 -7817.985} C_VEL
LIN {X 0,Y 461.871,Z 418.308,A -85,B 0,C 180,E1 -7818.369,E2 -7818.369} C_VEL
LIN {X 0,Y 461.535,Z 428.361,A -85,B 0,C 180,E1 -7818.916,E2 -7818.916} C_VEL
LIN {X 0,Y 461.153,Z 438.794,A -85,B 0,C 180,E1 -7819.685,E2 -7819.685} C_VEL
LIN {X 0,Y 460.776,Z 446.953,A -85,B 0,C 180,E1 -7820.452,E2 -7820.452} C_VEL
LIN {X 0,Y 460.484,Z 453.685,A -85,B 0,C 180,E1 -7821.221,E2 -7821.221} C_VEL
LIN {X 0,Y 460.229,Z 460.06,A -85,B 0,C 180,E1 -7822.101,E2 -7822.101} C_VEL
LIN {X 0,Y 460.068,Z 465.36,A -85,B 0,C 180,E1 -7822.981,E2 -7822.981} C_VEL
LIN {X 0,Y 459.908,Z 469.787,A -85,B 0,C 180,E1 -7823.86,E2 -7823.86} C_VEL
LIN {X 0,Y 459.675,Z 474.991,A -85,B 0,C 180,E1 -7825.176,E2 -7825.176} C_VEL
LIN {X 0,Y 459.659,Z 477.666,A -85,B 0,C 180,E1 -7826.055,E2 -7826.055} C_VEL
LIN {X 0,Y 459.592,Z 480.594,A -85,B 0,C 180,E1 -7827.371,E2 -7827.371} C_VEL
LIN {X 0,Y 459.52,Z 481.877,A -85,B 0,C 180,E1 -7828.247,E2 -7828.247} C_VEL
LIN {X 0,Y 459.492,Z 482.688,A -85,B 0,C 180,E1 -7829.124,E2 -7829.124} C_VEL
LIN {X 0,Y 459.472,Z 482.997,A -85,B 0,C 180,E1 -7830,E2 -7830} C_VEL
LIN {X 0,Y 459.493,Z 482.722,A -85,B 0,C 180,E1 -7830.876,E2 -7830.876} C_VEL
LIN {X 0,Y 459.517,Z 481.978,A -85,B 0,C 180,E1 -7831.753,E2 -7831.753} C_VEL
LIN {X 0,Y 459.577,Z 480.764,A -85,B 0,C 180,E1 -7832.629,E2 -7832.629} C_VEL
LIN {X 0,Y 459.655,Z 477.907,A -85,B 0,C 180,E1 -7833.945,E2 -7833.945} C_VEL
LIN {X 0,Y 459.671,Z 475.308,A -85,B 0,C 180,E1 -7834.824,E2 -7834.824} C_VEL
LIN {X 0,Y 459.898,Z 470.188,A -85,B 0,C 180,E1 -7836.141,E2 -7836.141} C_VEL
LIN {X 0,Y 460.113,Z 463.467,A -85,B 0,C 180,E1 -7837.46,E2 -7837.46} C_VEL
LIN {X 0,Y 460.387,Z 456.093,A -85,B 0,C 180,E1 -7838.559,E2 -7838.559} C_VEL
LIN {X 0,Y 460.729,Z 448.816,A -85,B 0,C 180,E1 -7839.438,E2 -7839.438} C_VEL
LIN {X 0,Y 461.005,Z 442.271,A -85,B 0,C 180,E1 -7840.097,E2 -7840.097} C_VEL
LIN {X 0,Y 461.311,Z 434.346,A -85,B 0,C 180,E1 -7840.756,E2 -7840.756} C_VEL
LIN {X 0,Y 461.614,Z 426.167,A -85,B 0,C 180,E1 -7841.304,E2 -7841.304} C_VEL
LIN {X 0,Y 461.894,Z 417.89,A -85,B 0,C 180,E1 -7841.742,E2 -7841.742} C_VEL
LIN {X 0,Y 462.077,Z 408.963,A -85,B 0,C 180,E1 -7842.099,E2 -7842.099} C_VEL
LIN {X 0,Y 462.297,Z 399.882,A -85,B 0,C 180,E1 -7842.346,E2 -7842.346} C_VEL
LIN {X 0,Y 462.623,Z 338.982,A -85,B 0,C 180,E1 -7843.312,E2 -7843.312} C_VEL
LIN {X 0,Y 460.52,Z 324.134,A -85,B 0,C 180,E1 -7843.628,E2 -7843.628} C_VEL
LIN {X 0,Y 460.478,Z 323.496,A -85,B 0,C 180,E1 -7843.686,E2 -7843.686} C_VEL
LIN {X 0,Y 460.952,Z 309.712,A -85,B 0,C 180,E1 -7846.839,E2 -7846.839} C_VEL
LIN {X 0,Y 461.414,Z 297.998,A -85,B 0,C 180,E1 -7849.578,E2 -7849.578} C_VEL
LIN {X 0,Y 461.26,Z 292.141,A -85,B 0,C 180,E1 -7850.98,E2 -7850.98} C_VEL
LIN {X 0,Y 460.581,Z 288.001,A -85,B 0,C 180,E1 -7852.07,E2 -7852.07} C_VEL
LIN {X 0,Y 460.521,Z 287.935,A -85,B 0,C 180,E1 -7855.296,E2 -7855.296} C_VEL
LIN {X 0,Y 460.505,Z 287.931,A -85,B 0,C 180,E1 -7858.235,E2 -7858.235} C_VEL
LIN {X 0,Y 460.518,Z 287.934,A -85,B 0,C 180,E1 -7861.282,E2 -7861.282} C_VEL
LIN {X 0,Y 460.518,Z 287.929,A -85,B 0,C 180,E1 -7864.503,E2 -7864.503} C_VEL
LIN {X 0,Y 460.494,Z 287.936,A -85,B 0,C 180,E1 -7867.623,E2 -7867.623} C_VEL
LIN {X 0,Y 460.51,Z 287.935,A -85,B 0,C 180,E1 -7871.012,E2 -7871.012} C_VEL
LIN {X 0,Y 460.505,Z 287.932,A -85,B 0,C 180,E1 -7874.589,E2 -7874.589} C_VEL
LIN {X 0,Y 460.468,Z 287.936,A -85,B 0,C 180,E1 -7877.812,E2 -7877.812} C_VEL
LIN {X 0,Y 460.506,Z 287.931,A -85,B 0,C 180,E1 -7880.135,E2 -7880.135} C_VEL
LIN {X 0,Y 460.465,Z 287.937,A -85,B 0,C 180,E1 -7883.469,E2 -7883.469} C_VEL
LIN {X 0,Y 460.508,Z 287.936,A -85,B 0,C 180,E1 -7886.673,E2 -7886.673} C_VEL
LIN {X 0,Y 460.493,Z 287.932,A -85,B 0,C 180,E1 -7889.759,E2 -7889.759} C_VEL
LIN {X 0,Y 460.483,Z 287.941,A -85,B 0,C 180,E1 -7892.75,E2 -7892.75} C_VEL
LIN {X 0,Y 460.508,Z 287.93,A -85,B 0,C 180,E1 -7895.666,E2 -7895.666} C_VEL
LIN {X 0,Y 460.509,Z 287.938,A -85,B 0,C 180,E1 -7898.579,E2 -7898.579} C_VEL
LIN {X 0,Y 460.571,Z 287.923,A -85,B 0,C 180,E1 -7901.31,E2 -7901.31} C_VEL
LIN {X 0,Y 460.537,Z 287.928,A -85,B 0,C 180,E1 -7904.964,E2 -7904.964} C_VEL
LIN {X 0,Y 460.597,Z 287.924,A -85,B 0,C 180,E1 -7908.559,E2 -7908.559} C_VEL
LIN {X 0,Y 460.605,Z 287.918,A -85,B 0,C 180,E1 -7911.223,E2 -7911.223} C_VEL
LIN {X 0,Y 460.659,Z 287.915,A -85,B 0,C 180,E1 -7913.869,E2 -7913.869} C_VEL
LIN {X 0,Y 460.744,Z 287.901,A -85,B 0,C 180,E1 -7917.377,E2 -7917.377} C_VEL
LIN {X 0,Y 460.807,Z 287.901,A -85,B 0,C 180,E1 -7920,E2 -7920} C_VEL
LIN {X 0,Y 460.743,Z 287.902,A -85,B 0,C 180,E1 -7922.623,E2 -7922.623} C_VEL
LIN {X 0,Y 460.657,Z 287.916,A -85,B 0,C 180,E1 -7926.131,E2 -7926.131} C_VEL
LIN {X 0,Y 460.576,Z 287.922,A -85,B 0,C 180,E1 -7928.777,E2 -7928.777} C_VEL
LIN {X 0,Y 460.586,Z 287.921,A -85,B 0,C 180,E1 -7932.435,E2 -7932.435} C_VEL
LIN {X 0,Y 460.547,Z 287.929,A -85,B 0,C 180,E1 -7935.979,E2 -7935.979} C_VEL
LIN {X 0,Y 460.549,Z 287.932,A -85,B 0,C 180,E1 -7939.616,E2 -7939.616} C_VEL
LIN {X 0,Y 460.485,Z 287.933,A -85,B 0,C 180,E1 -7942.43,E2 -7942.43} C_VEL
LIN {X 0,Y 460.525,Z 287.931,A -85,B 0,C 180,E1 -7945.793,E2 -7945.793} C_VEL
LIN {X 0,Y 460.509,Z 287.937,A -85,B 0,C 180,E1 -7949.233,E2 -7949.233} C_VEL
LIN {X 0,Y 460.508,Z 287.93,A -85,B 0,C 180,E1 -7952.286,E2 -7952.286} C_VEL
LIN {X 0,Y 460.496,Z 287.936,A -85,B 0,C 180,E1 -7955.447,E2 -7955.447} C_VEL
LIN {X 0,Y 460.495,Z 287.938,A -85,B 0,C 180,E1 -7958.892,E2 -7958.892} C_VEL
LIN {X 0,Y 460.494,Z 287.933,A -85,B 0,C 180,E1 -7961.599,E2 -7961.599} C_VEL
LIN {X 0,Y 460.504,Z 287.935,A -85,B 0,C 180,E1 -7964.59,E2 -7964.59} C_VEL
LIN {X 0,Y 460.468,Z 287.935,A -85,B 0,C 180,E1 -7967.814,E2 -7967.814} C_VEL
LIN {X 0,Y 460.504,Z 287.932,A -85,B 0,C 180,E1 -7970.136,E2 -7970.136} C_VEL
LIN {X 0,Y 460.465,Z 287.936,A -85,B 0,C 180,E1 -7973.47,E2 -7973.47} C_VEL
LIN {X 0,Y 460.512,Z 287.937,A -85,B 0,C 180,E1 -7976.675,E2 -7976.675} C_VEL
LIN {X 0,Y 460.498,Z 287.932,A -85,B 0,C 180,E1 -7979.76,E2 -7979.76} C_VEL
LIN {X 0,Y 460.487,Z 287.937,A -85,B 0,C 180,E1 -7982.751,E2 -7982.751} C_VEL
LIN {X 0,Y 460.514,Z 287.933,A -85,B 0,C 180,E1 -7985.667,E2 -7985.667} C_VEL
LIN {X 0,Y 460.593,Z 288.114,A -85,B 0,C 180,E1 -7988.049,E2 -7988.049} C_VEL
LIN {X 0,Y 461.437,Z 293.906,A -85,B 0,C 180,E1 -7989.495,E2 -7989.495} C_VEL
LIN {X 0,Y 461.184,Z 303.665,A -85,B 0,C 180,E1 -7991.796,E2 -7991.796} C_VEL
LIN {X 0,Y 460.658,Z 317.328,A -85,B 0,C 180,E1 -7994.968,E2 -7994.968} C_VEL
LIN {X 0,Y 460.496,Z 323.682,A -85,B 0,C 180,E1 -7996.385,E2 -7996.385} C_VEL
LIN {X 0,Y 461.1,Z 327.902,A -85,B 0,C 180,E1 -7996.515,E2 -7996.515} C_VEL
LIN {X 0,Y 462.663,Z 338.587,A -85,B 0,C 180,E1 -7996.728,E2 -7996.728} C_VEL
LIN {X 0,Y 462.27,Z 399.641,A -85,B 0,C 180,E1 -7997.693,E2 -7997.693} C_VEL
LIN {X 0,Y 462.061,Z 409.282,A -85,B 0,C 180,E1 -7997.956,E2 -7997.956} C_VEL
LIN {X 0,Y 461.911,Z 419.33,A -85,B 0,C 180,E1 -7998.37,E2 -7998.37} C_VEL
LIN {X 0,Y 461.466,Z 430.737,A -85,B 0,C 180,E1 -7999.026,E2 -7999.026} C_VEL
LIN {X 0,Y 461.135,Z 439.314,A -85,B 0,C 180,E1 -7999.684,E2 -7999.684} C_VEL
LIN {X 0,Y 460.783,Z 447.381,A -85,B 0,C 180,E1 -8000.453,E2 -8000.453} C_VEL
LIN {X 0,Y 460.459,Z 454.042,A -85,B 0,C 180,E1 -8001.221,E2 -8001.221} C_VEL
LIN {X 0,Y 460.203,Z 460.364,A -85,B 0,C 180,E1 -8002.1,E2 -8002.1} C_VEL
LIN {X 0,Y 460.028,Z 465.615,A -85,B 0,C 180,E1 -8002.98,E2 -8002.98} C_VEL
LIN {X 0,Y 459.911,Z 469.993,A -85,B 0,C 180,E1 -8003.86,E2 -8003.86} C_VEL
LIN {X 0,Y 459.672,Z 475.153,A -85,B 0,C 180,E1 -8005.176,E2 -8005.176} C_VEL
LIN {X 0,Y 459.638,Z 478.94,A -85,B 0,C 180,E1 -8006.494,E2 -8006.494} C_VEL
LIN {X 0,Y 459.591,Z 480.681,A -85,B 0,C 180,E1 -8007.371,E2 -8007.371} C_VEL
LIN {X 0,Y 459.519,Z 481.929,A -85,B 0,C 180,E1 -8008.247,E2 -8008.247} C_VEL
LIN {X 0,Y 459.492,Z 482.706,A -85,B 0,C 180,E1 -8009.124,E2 -8009.124} C_VEL
LIN {X 0,Y 459.471,Z 483,A -85,B 0,C 180,E1 -8010,E2 -8010} C_VEL
LIN {X 0,Y 459.492,Z 482.705,A -85,B 0,C 180,E1 -8010.876,E2 -8010.876} C_VEL
LIN {X 0,Y 459.519,Z 481.926,A -85,B 0,C 180,E1 -8011.753,E2 -8011.753} C_VEL
LIN {X 0,Y 459.591,Z 480.677,A -85,B 0,C 180,E1 -8012.629,E2 -8012.629} C_VEL
LIN {X 0,Y 459.656,Z 477.784,A -85,B 0,C 180,E1 -8013.945,E2 -8013.945} C_VEL
LIN {X 0,Y 459.672,Z 475.146,A -85,B 0,C 180,E1 -8014.824,E2 -8014.824} C_VEL
LIN {X 0,Y 459.907,Z 469.982,A -85,B 0,C 180,E1 -8016.14,E2 -8016.14} C_VEL
LIN {X 0,Y 460.124,Z 463.177,A -85,B 0,C 180,E1 -8017.46,E2 -8017.46} C_VEL
LIN {X 0,Y 460.387,Z 455.733,A -85,B 0,C 180,E1 -8018.559,E2 -8018.559} C_VEL
LIN {X 0,Y 460.733,Z 448.389,A -85,B 0,C 180,E1 -8019.438,E2 -8019.438} C_VEL
LIN {X 0,Y 461.057,Z 440.523,A -85,B 0,C 180,E1 -8020.207,E2 -8020.207} C_VEL
LIN {X 0,Y 461.412,Z 432.21,A -85,B 0,C 180,E1 -8020.864,E2 -8020.864} C_VEL
LIN {X 0,Y 461.771,Z 421.594,A -85,B 0,C 180,E1 -8021.523,E2 -8021.523} C_VEL
LIN {X 0,Y 462.06,Z 410.051,A -85,B 0,C 180,E1 -8022.016,E2 -8022.016} C_VEL
LIN {X 0,Y 462.264,Z 400.399,A -85,B 0,C 180,E1 -8022.289,E2 -8022.289} C_VEL
LIN {X 0,Y 462.515,Z 337.228,A -85,B 0,C 180,E1 -8023.295,E2 -8023.295} C_VEL
LIN {X 0,Y 460.5,Z 323.932,A -85,B 0,C 180,E1 -8023.59,E2 -8023.59} C_VEL
LIN {X 0,Y 460.518,Z 321.22,A -85,B 0,C 180,E1 -8024.133,E2 -8024.133} C_VEL
LIN {X 0,Y 461.028,Z 307.555,A -85,B 0,C 180,E1 -8027.293,E2 -8027.293} C_VEL
LIN {X 0,Y 461.469,Z 295.843,A -85,B 0,C 180,E1 -8030.039,E2 -8030.039} C_VEL
LIN {X 0,Y 460.882,Z 289.699,A -85,B 0,C 180,E1 -8031.536,E2 -8031.536} C_VEL
LIN {X 0,Y 460.546,Z 288.014,A -85,B 0,C 180,E1 -8032.013,E2 -8032.013} C_VEL
LIN {X 0,Y 460.514,Z 287.933,A -85,B 0,C 180,E1 -8034.333,E2 -8034.333} C_VEL
LIN {X 0,Y 460.488,Z 287.937,A -85,B 0,C 180,E1 -8037.249,E2 -8037.249} C_VEL
LIN {X 0,Y 460.498,Z 287.932,A -85,B 0,C 180,E1 -8040.24,E2 -8040.24} C_VEL
LIN {X 0,Y 460.512,Z 287.937,A -85,B 0,C 180,E1 -8043.325,E2 -8043.325} C_VEL
LIN {X 0,Y 460.466,Z 287.936,A -85,B 0,C 180,E1 -8046.529,E2 -8046.529} C_VEL
LIN {X 0,Y 460.507,Z 287.931,A -85,B 0,C 180,E1 -8049.864,E2 -8049.864} C_VEL
LIN {X 0,Y 460.456,Z 287.941,A -85,B 0,C 180,E1 -8052.893,E2 -8052.893} C_VEL
LIN {X 0,Y 460.496,Z 287.932,A -85,B 0,C 180,E1 -8055.831,E2 -8055.831} C_VEL
LIN {X 0,Y 460.507,Z 287.938,A -85,B 0,C 180,E1 -8058.986,E2 -8058.986} C_VEL
LIN {X 0,Y 460.49,Z 287.934,A -85,B 0,C 180,E1 -8062.376,E2 -8062.376} C_VEL
LIN {X 0,Y 460.526,Z 287.928,A -85,B 0,C 180,E1 -8065.622,E2 -8065.622} C_VEL
LIN {X 0,Y 460.495,Z 287.939,A -85,B 0,C 180,E1 -8068.741,E2 -8068.741} C_VEL
LIN {X 0,Y 460.497,Z 287.932,A -85,B 0,C 180,E1 -8071.763,E2 -8071.763} C_VEL
LIN {X 0,Y 460.512,Z 287.937,A -85,B 0,C 180,E1 -8074.703,E2 -8074.703} C_VEL
LIN {X 0,Y 460.493,Z 287.932,A -85,B 0,C 180,E1 -8077.571,E2 -8077.571} C_VEL
LIN {X 0,Y 460.55,Z 287.931,A -85,B 0,C 180,E1 -8080.384,E2 -8080.384} C_VEL
LIN {X 0,Y 460.556,Z 287.928,A -85,B 0,C 180,E1 -8084.057,E2 -8084.057} C_VEL
LIN {X 0,Y 460.599,Z 287.92,A -85,B 0,C 180,E1 -8087.666,E2 -8087.666} C_VEL
LIN {X 0,Y 460.597,Z 287.919,A -85,B 0,C 180,E1 -8091.223,E2 -8091.223} C_VEL
LIN {X 0,Y 460.658,Z 287.916,A -85,B 0,C 180,E1 -8093.869,E2 -8093.869} C_VEL
LIN {X 0,Y 460.744,Z 287.901,A -85,B 0,C 180,E1 -8097.377,E2 -8097.377} C_VEL
LIN {X 0,Y 460.807,Z 287.901,A -85,B 0,C 180,E1 -8100,E2 -8100} C_VEL
LIN {X 0,Y 460.744,Z 287.902,A -85,B 0,C 180,E1 -8102.623,E2 -8102.623} C_VEL
LIN {X 0,Y 460.657,Z 287.916,A -85,B 0,C 180,E1 -8106.131,E2 -8106.131} C_VEL
LIN {X 0,Y 460.573,Z 287.922,A -85,B 0,C 180,E1 -8108.777,E2 -8108.777} C_VEL
LIN {X 0,Y 460.587,Z 287.921,A -85,B 0,C 180,E1 -8112.435,E2 -8112.435} C_VEL
LIN {X 0,Y 460.547,Z 287.929,A -85,B 0,C 180,E1 -8115.979,E2 -8115.979} C_VEL
LIN {X 0,Y 460.549,Z 287.932,A -85,B 0,C 180,E1 -8119.616,E2 -8119.616} C_VEL
LIN {X 0,Y 460.486,Z 287.933,A -85,B 0,C 180,E1 -8122.43,E2 -8122.43} C_VEL
LIN {X 0,Y 460.525,Z 287.931,A -85,B 0,C 180,E1 -8125.794,E2 -8125.794} C_VEL
LIN {X 0,Y 460.505,Z 287.938,A -85,B 0,C 180,E1 -8129.233,E2 -8129.233} C_VEL
LIN {X 0,Y 460.506,Z 287.93,A -85,B 0,C 180,E1 -8132.286,E2 -8132.286} C_VEL
LIN {X 0,Y 460.497,Z 287.936,A -85,B 0,C 180,E1 -8135.447,E2 -8135.447} C_VEL
LIN {X 0,Y 460.487,Z 287.938,A -85,B 0,C 180,E1 -8138.89,E2 -8138.89} C_VEL
LIN {X 0,Y 460.495,Z 287.933,A -85,B 0,C 180,E1 -8141.599,E2 -8141.599} C_VEL
LIN {X 0,Y 460.505,Z 287.934,A -85,B 0,C 180,E1 -8144.59,E2 -8144.59} C_VEL
LIN {X 0,Y 460.469,Z 287.935,A -85,B 0,C 180,E1 -8147.814,E2 -8147.814} C_VEL
LIN {X 0,Y 460.505,Z 287.931,A -85,B 0,C 180,E1 -8150.136,E2 -8150.136} C_VEL
LIN {X 0,Y 460.466,Z 287.936,A -85,B 0,C 180,E1 -8153.471,E2 -8153.471} C_VEL
LIN {X 0,Y 460.513,Z 287.937,A -85,B 0,C 180,E1 -8156.675,E2 -8156.675} C_VEL
LIN {X 0,Y 460.48,Z 287.934,A -85,B 0,C 180,E1 -8159.759,E2 -8159.759} C_VEL
LIN {X 0,Y 460.488,Z 287.937,A -85,B 0,C 180,E1 -8162.751,E2 -8162.751} C_VEL
LIN {X 0,Y 460.513,Z 287.933,A -85,B 0,C 180,E1 -8165.667,E2 -8165.667} C_VEL
LIN {X 0,Y 460.565,Z 288.068,A -85,B 0,C 180,E1 -8168.08,E2 -8168.08} C_VEL
LIN {X 0,Y 461.396,Z 293.703,A -85,B 0,C 180,E1 -8169.493,E2 -8169.493} C_VEL
LIN {X 0,Y 461.186,Z 303.461,A -85,B 0,C 180,E1 -8171.797,E2 -8171.797} C_VEL
LIN {X 0,Y 460.66,Z 317.122,A -85,B 0,C 180,E1 -8174.968,E2 -8174.968} C_VEL
LIN {X 0,Y 460.563,Z 319.641,A -85,B 0,C 180,E1 -8175.548,E2 -8175.548} C_VEL
LIN {X 0,Y 460.294,Z 322.009,A -85,B 0,C 180,E1 -8175.918,E2 -8175.918} C_VEL
LIN {X 0,Y 459.734,Z 325.111,A -85,B 0,C 180,E1 -8176.194,E2 -8176.194} C_VEL
LIN {X 0,Y 458.599,Z 330.524,A -85,B 0,C 180,E1 -8176.461,E2 -8176.461} C_VEL
LIN {X 0,Y 457.278,Z 336.568,A -85,B 0,C 180,E1 -8176.585,E2 -8176.585} C_VEL
LIN {X 0,Y 455.93,Z 345.006,A -85,B 0,C 180,E1 -8176.677,E2 -8176.677} C_VEL
LIN {X 0,Y 455.684,Z 349.261,A -85,B 0,C 180,E1 -8176.738,E2 -8176.738} C_VEL
LIN {X 0,Y 455.423,Z 399.621,A -85,B 0,C 180,E1 -8177.552,E2 -8177.552} C_VEL
LIN {X 0,Y 455.184,Z 408.72,A -85,B 0,C 180,E1 -8177.8,E2 -8177.8} C_VEL
LIN {X 0,Y 454.919,Z 418.318,A -85,B 0,C 180,E1 -8178.188,E2 -8178.188} C_VEL
LIN {X 0,Y 454.577,Z 428.369,A -85,B 0,C 180,E1 -8178.745,E2 -8178.745} C_VEL
LIN {X 0,Y 454.16,Z 438.799,A -85,B 0,C 180,E1 -8179.524,E2 -8179.524} C_VEL
LIN {X 0,Y 453.774,Z 446.957,A -85,B 0,C 180,E1 -8180.304,E2 -8180.304} C_VEL
LIN {X 0,Y 453.469,Z 453.689,A -85,B 0,C 180,E1 -8181.084,E2 -8181.084} C_VEL
LIN {X 0,Y 453.172,Z 460.063,A -85,B 0,C 180,E1 -8181.977,E2 -8181.977} C_VEL
LIN {X 0,Y 452.957,Z 466.41,A -85,B 0,C 180,E1 -8183.07,E2 -8183.07} C_VEL
LIN {X 0,Y 452.776,Z 471.701,A -85,B 0,C 180,E1 -8184.21,E2 -8184.21} C_VEL
LIN {X 0,Y 452.547,Z 476.485,A -85,B 0,C 180,E1 -8185.547,E2 -8185.547} C_VEL
LIN {X 0,Y 452.543,Z 478.818,A -85,B 0,C 180,E1 -8186.439,E2 -8186.439} C_VEL
LIN {X 0,Y 452.517,Z 480.595,A -85,B 0,C 180,E1 -8187.33,E2 -8187.33} C_VEL
LIN {X 0,Y 452.436,Z 481.877,A -85,B 0,C 180,E1 -8188.22,E2 -8188.22} C_VEL
LIN {X 0,Y 452.401,Z 482.689,A -85,B 0,C 180,E1 -8189.11,E2 -8189.11} C_VEL
LIN {X 0,Y 452.38,Z 482.997,A -85,B 0,C 180,E1 -8190,E2 -8190} C_VEL
LIN {X 0,Y 452.401,Z 482.722,A -85,B 0,C 180,E1 -8190.89,E2 -8190.89} C_VEL
LIN {X 0,Y 452.433,Z 481.978,A -85,B 0,C 180,E1 -8191.78,E2 -8191.78} C_VEL
LIN {X 0,Y 452.504,Z 480.764,A -85,B 0,C 180,E1 -8192.671,E2 -8192.671} C_VEL
LIN {X 0,Y 452.552,Z 477.906,A -85,B 0,C 180,E1 -8194.007,E2 -8194.007} C_VEL
LIN {X 0,Y 452.605,Z 475.307,A -85,B 0,C 180,E1 -8194.899,E2 -8194.899} C_VEL
LIN {X 0,Y 452.824,Z 470.186,A -85,B 0,C 180,E1 -8196.237,E2 -8196.237} C_VEL
LIN {X 0,Y 453.021,Z 464.679,A -85,B 0,C 180,E1 -8197.353,E2 -8197.353} C_VEL
LIN {X 0,Y 453.287,Z 457.768,A -85,B 0,C 180,E1 -8198.47,E2 -8198.47} C_VEL
LIN {X 0,Y 453.692,Z 449.832,A -85,B 0,C 180,E1 -8199.473,E2 -8199.473} C_VEL
LIN {X 0,Y 454.021,Z 442.266,A -85,B 0,C 180,E1 -8200.254,E2 -8200.254} C_VEL
LIN {X 0,Y 454.353,Z 434.34,A -85,B 0,C 180,E1 -8200.922,E2 -8200.922} C_VEL
LIN {X 0,Y 454.662,Z 426.16,A -85,B 0,C 180,E1 -8201.479,E2 -8201.479} C_VEL
LIN {X 0,Y 454.962,Z 417.88,A -85,B 0,C 180,E1 -8201.923,E2 -8201.923} C_VEL
LIN {X 0,Y 455.164,Z 408.95,A -85,B 0,C 180,E1 -8202.286,E2 -8202.286} C_VEL
LIN {X 0,Y 455.381,Z 399.963,A -85,B 0,C 180,E1 -8202.535,E2 -8202.535} C_VEL
LIN {X 0,Y 455.735,Z 339.997,A -85,B 0,C 180,E1 -8203.5,E2 -8203.5} C_VEL
LIN {X 0,Y 453.516,Z 324.228,A -85,B 0,C 180,E1 -8203.838,E2 -8203.838} C_VEL
LIN {X 0,Y 453.437,Z 323.073,A -85,B 0,C 180,E1 -8203.985,E2 -8203.985} C_VEL
LIN {X 0,Y 453.956,Z 309.71,A -85,B 0,C 180,E1 -8207.106,E2 -8207.106} C_VEL
LIN {X 0,Y 454.438,Z 297.996,A -85,B 0,C 180,E1 -8209.891,E2 -8209.891} C_VEL
LIN {X 0,Y 454.138,Z 292.372,A -85,B 0,C 180,E1 -8211.269,E2 -8211.269} C_VEL
LIN {X 0,Y 453.523,Z 288.893,A -85,B 0,C 180,E1 -8212.192,E2 -8212.192} C_VEL
LIN {X 0,Y 453.468,Z 288.81,A -85,B 0,C 180,E1 -8214.736,E2 -8214.736} C_VEL
LIN {X 0,Y 453.461,Z 288.811,A -85,B 0,C 180,E1 -8217.942,E2 -8217.942} C_VEL
LIN {X 0,Y 453.472,Z 288.807,A -85,B 0,C 180,E1 -8220.759,E2 -8220.759} C_VEL
LIN {X 0,Y 453.463,Z 288.81,A -85,B 0,C 180,E1 -8223.913,E2 -8223.913} C_VEL
LIN {X 0,Y 453.445,Z 288.816,A -85,B 0,C 180,E1 -8227.189,E2 -8227.189} C_VEL
LIN {X 0,Y 453.465,Z 288.808,A -85,B 0,C 180,E1 -8230.611,E2 -8230.611} C_VEL
LIN {X 0,Y 453.475,Z 288.807,A -85,B 0,C 180,E1 -8234.528,E2 -8234.528} C_VEL
LIN {X 0,Y 453.429,Z 288.812,A -85,B 0,C 180,E1 -8238.07,E2 -8238.07} C_VEL
LIN {X 0,Y 453.458,Z 288.814,A -85,B 0,C 180,E1 -8240.797,E2 -8240.797} C_VEL
LIN {X 0,Y 453.443,Z 288.81,A -85,B 0,C 180,E1 -8243.916,E2 -8243.916} C_VEL
LIN {X 0,Y 453.465,Z 288.811,A -85,B 0,C 180,E1 -8247.15,E2 -8247.15} C_VEL
LIN {X 0,Y 453.452,Z 288.811,A -85,B 0,C 180,E1 -8250.267,E2 -8250.267} C_VEL
LIN {X 0,Y 453.433,Z 288.813,A -85,B 0,C 180,E1 -8253.289,E2 -8253.289} C_VEL
LIN {X 0,Y 453.482,Z 288.809,A -85,B 0,C 180,E1 -8256.238,E2 -8256.238} C_VEL
LIN {X 0,Y 453.464,Z 288.809,A -85,B 0,C 180,E1 -8259.117,E2 -8259.117} C_VEL
LIN {X 0,Y 453.472,Z 288.808,A -85,B 0,C 180,E1 -8261.943,E2 -8261.943} C_VEL
LIN {X 0,Y 453.508,Z 288.806,A -85,B 0,C 180,E1 -8264.725,E2 -8264.725} C_VEL
LIN {X 0,Y 453.547,Z 288.804,A -85,B 0,C 180,E1 -8268.379,E2 -8268.379} C_VEL
LIN {X 0,Y 453.572,Z 288.794,A -85,B 0,C 180,E1 -8271.086,E2 -8271.086} C_VEL
LIN {X 0,Y 453.627,Z 288.79,A -85,B 0,C 180,E1 -8273.774,E2 -8273.774} C_VEL
LIN {X 0,Y 453.691,Z 288.78,A -85,B 0,C 180,E1 -8277.336,E2 -8277.336} C_VEL
LIN {X 0,Y 453.756,Z 288.779,A -85,B 0,C 180,E1 -8280,E2 -8280} C_VEL
LIN {X 0,Y 453.69,Z 288.78,A -85,B 0,C 180,E1 -8282.664,E2 -8282.664} C_VEL
LIN {X 0,Y 453.625,Z 288.791,A -85,B 0,C 180,E1 -8286.226,E2 -8286.226} C_VEL
LIN {X 0,Y 453.546,Z 288.797,A -85,B 0,C 180,E1 -8288.914,E2 -8288.914} C_VEL
LIN {X 0,Y 453.554,Z 288.797,A -85,B 0,C 180,E1 -8292.529,E2 -8292.529} C_VEL
LIN {X 0,Y 453.49,Z 288.806,A -85,B 0,C 180,E1 -8296.198,E2 -8296.198} C_VEL
LIN {X 0,Y 453.507,Z 288.804,A -85,B 0,C 180,E1 -8299.039,E2 -8299.039} C_VEL
LIN {X 0,Y 453.461,Z 288.811,A -85,B 0,C 180,E1 -8301.837,E2 -8301.837} C_VEL
LIN {X 0,Y 453.458,Z 288.809,A -85,B 0,C 180,E1 -8304.738,E2 -8304.738} C_VEL
LIN {X 0,Y 453.452,Z 288.81,A -85,B 0,C 180,E1 -8307.943,E2 -8307.943} C_VEL
LIN {X 0,Y 453.447,Z 288.812,A -85,B 0,C 180,E1 -8310.762,E2 -8310.762} C_VEL
LIN {X 0,Y 453.457,Z 288.809,A -85,B 0,C 180,E1 -8313.914,E2 -8313.914} C_VEL
LIN {X 0,Y 453.44,Z 288.817,A -85,B 0,C 180,E1 -8317.191,E2 -8317.191} C_VEL
LIN {X 0,Y 453.462,Z 288.811,A -85,B 0,C 180,E1 -8320.612,E2 -8320.612} C_VEL
LIN {X 0,Y 453.474,Z 288.81,A -85,B 0,C 180,E1 -8324.529,E2 -8324.529} C_VEL
LIN {X 0,Y 453.429,Z 288.812,A -85,B 0,C 180,E1 -8328.072,E2 -8328.072} C_VEL
LIN {X 0,Y 453.435,Z 288.819,A -85,B 0,C 180,E1 -8330.802,E2 -8330.802} C_VEL
LIN {X 0,Y 453.444,Z 288.811,A -85,B 0,C 180,E1 -8333.917,E2 -8333.917} C_VEL
LIN {X 0,Y 453.47,Z 288.809,A -85,B 0,C 180,E1 -8337.151,E2 -8337.151} C_VEL
LIN {X 0,Y 453.457,Z 288.813,A -85,B 0,C 180,E1 -8340.268,E2 -8340.268} C_VEL
LIN {X 0,Y 453.438,Z 288.811,A -85,B 0,C 180,E1 -8343.29,E2 -8343.29} C_VEL
LIN {X 0,Y 453.489,Z 288.796,A -85,B 0,C 180,E1 -8346.239,E2 -8346.239} C_VEL
LIN {X 0,Y 453.542,Z 288.975,A -85,B 0,C 180,E1 -8347.898,E2 -8347.898} C_VEL
LIN {X 0,Y 454.47,Z 295.859,A -85,B 0,C 180,E1 -8349.639,E2 -8349.639} C_VEL
LIN {X 0,Y 454.124,Z 305.618,A -85,B 0,C 180,E1 -8351.97,E2 -8351.97} C_VEL
LIN {X 0,Y 453.567,Z 319.281,A -85,B 0,C 180,E1 -8355.187,E2 -8355.187} C_VEL
LIN {X 0,Y 453.453,Z 323.707,A -85,B 0,C 180,E1 -8356.172,E2 -8356.172} C_VEL
LIN {X 0,Y 454.143,Z 328.079,A -85,B 0,C 180,E1 -8356.307,E2 -8356.307} C_VEL
LIN {X 0,Y 455.81,Z 340.246,A -85,B 0,C 180,E1 -8356.551,E2 -8356.551} C_VEL
LIN {X 0,Y 455.353,Z 399.692,A -85,B 0,C 180,E1 -8357.504,E2 -8357.504} C_VEL
LIN {X 0,Y 455.131,Z 409.29,A -85,B 0,C 180,E1 -8357.77,E2 -8357.77} C_VEL
LIN {X 0,Y 454.962,Z 419.336,A -85,B 0,C 180,E1 -8358.19,E2 -8358.19} C_VEL
LIN {X 0,Y 454.496,Z 430.741,A -85,B 0,C 180,E1 -8358.855,E2 -8358.855} C_VEL
LIN {X 0,Y 454.139,Z 439.317,A -85,B 0,C 180,E1 -8359.524,E2 -8359.524} C_VEL
LIN {X 0,Y 453.764,Z 447.383,A -85,B 0,C 180,E1 -8360.303,E2 -8360.303} C_VEL
LIN {X 0,Y 453.445,Z 454.044,A -85,B 0,C 180,E1 -8361.084,E2 -8361.084} C_VEL
LIN {X 0,Y 453.151,Z 460.365,A -85,B 0,C 180,E1 -8361.976,E2 -8361.976} C_VEL
LIN {X 0,Y 452.969,Z 465.616,A -85,B 0,C 180,E1 -8362.87,E2 -8362.87} C_VEL
LIN {X 0,Y 452.836,Z 469.994,A -85,B 0,C 180,E1 -8363.763,E2 -8363.763} C_VEL
LIN {X 0,Y 452.606,Z 475.154,A -85,B 0,C 180,E1 -8365.101,E2 -8365.101} C_VEL
LIN {X 0,Y 452.541,Z 478.941,A -85,B 0,C 180,E1 -8366.439,E2 -8366.439} C_VEL
LIN {X 0,Y 452.516,Z 480.682,A -85,B 0,C 180,E1 -8367.33,E2 -8367.33} C_VEL
LIN {X 0,Y 452.435,Z 481.929,A -85,B 0,C 180,E1 -8368.22,E2 -8368.22} C_VEL
LIN {X 0,Y 452.4,Z 482.706,A -85,B 0,C 180,E1 -8369.11,E2 -8369.11} C_VEL
LIN {X 0,Y 452.378,Z 483,A -85,B 0,C 180,E1 -8370,E2 -8370} C_VEL
LIN {X 0,Y 452.4,Z 482.705,A -85,B 0,C 180,E1 -8370.89,E2 -8370.89} C_VEL
LIN {X 0,Y 452.435,Z 481.926,A -85,B 0,C 180,E1 -8371.78,E2 -8371.78} C_VEL
LIN {X 0,Y 452.516,Z 480.677,A -85,B 0,C 180,E1 -8372.67,E2 -8372.67} C_VEL
LIN {X 0,Y 452.553,Z 477.783,A -85,B 0,C 180,E1 -8374.007,E2 -8374.007} C_VEL
LIN {X 0,Y 452.606,Z 475.145,A -85,B 0,C 180,E1 -8374.899,E2 -8374.899} C_VEL
LIN {X 0,Y 452.83,Z 469.981,A -85,B 0,C 180,E1 -8376.237,E2 -8376.237} C_VEL
LIN {X 0,Y 453.072,Z 463.175,A -85,B 0,C 180,E1 -8377.576,E2 -8377.576} C_VEL
LIN {X 0,Y 453.362,Z 455.731,A -85,B 0,C 180,E1 -8378.693,E2 -8378.693} C_VEL
LIN {X 0,Y 453.713,Z 448.387,A -85,B 0,C 180,E1 -8379.585,E2 -8379.585} C_VEL
LIN {X 0,Y 454.074,Z 440.52,A -85,B 0,C 180,E1 -8380.365,E2 -8380.365} C_VEL
LIN {X 0,Y 454.447,Z 432.206,A -85,B 0,C 180,E1 -8381.033,E2 -8381.033} C_VEL
LIN {X 0,Y 454.829,Z 421.589,A -85,B 0,C 180,E1 -8381.701,E2 -8381.701} C_VEL
LIN {X 0,Y 455.115,Z 410.043,A -85,B 0,C 180,E1 -8382.202,E2 -8382.202} C_VEL
LIN {X 0,Y 455.343,Z 400.386,A -85,B 0,C 180,E1 -8382.479,E2 -8382.479} C_VEL
LIN {X 0,Y 455.696,Z 338.463,A -85,B 0,C 180,E1 -8383.478,E2 -8383.478} C_VEL
LIN {X 0,Y 453.47,Z 323.929,A -85,B 0,C 180,E1 -8383.805,E2 -8383.805} C_VEL
LIN {X 0,Y 453.513,Z 321.219,A -85,B 0,C 180,E1 -8384.356,E2 -8384.356} C_VEL
LIN {X 0,Y 454.033,Z 307.554,A -85,B 0,C 180,E1 -8387.568,E2 -8387.568} C_VEL
LIN {X 0,Y 454.435,Z 297.793,A -85,B 0,C 180,E1 -8389.891,E2 -8389.891} C_VEL
LIN {X 0,Y 454.099,Z 292.189,A -85,B 0,C 180,E1 -8391.266,E2 -8391.266} C_VEL
LIN {X 0,Y 453.523,Z 288.903,A -85,B 0,C 180,E1 -8392.132,E2 -8392.132} C_VEL
LIN {X 0,Y 453.466,Z 288.811,A -85,B 0,C 180,E1 -8394.737,E2 -8394.737} C_VEL
LIN {X 0,Y 453.459,Z 288.811,A -85,B 0,C 180,E1 -8397.942,E2 -8397.942} C_VEL
LIN {X 0,Y 453.453,Z 288.81,A -85,B 0,C 180,E1 -8400.76,E2 -8400.76} C_VEL
LIN {X 0,Y 453.461,Z 288.81,A -85,B 0,C 180,E1 -8403.913,E2 -8403.913} C_VEL
LIN {X 0,Y 453.443,Z 288.817,A -85,B 0,C 180,E1 -8407.19,E2 -8407.19} C_VEL
LIN {X 0,Y 453.464,Z 288.809,A -85,B 0,C 180,E1 -8410.611,E2 -8410.611} C_VEL
LIN {X 0,Y 453.474,Z 288.808,A -85,B 0,C 180,E1 -8414.528,E2 -8414.528} C_VEL
LIN {X 0,Y 453.428,Z 288.812,A -85,B 0,C 180,E1 -8418.07,E2 -8418.07} C_VEL
LIN {X 0,Y 453.439,Z 288.816,A -85,B 0,C 180,E1 -8420.8,E2 -8420.8} C_VEL
LIN {X 0,Y 453.441,Z 288.81,A -85,B 0,C 180,E1 -8423.916,E2 -8423.916} C_VEL
LIN {X 0,Y 453.464,Z 288.811,A -85,B 0,C 180,E1 -8427.15,E2 -8427.15} C_VEL
LIN {X 0,Y 453.451,Z 288.811,A -85,B 0,C 180,E1 -8430.267,E2 -8430.267} C_VEL
LIN {X 0,Y 453.432,Z 288.813,A -85,B 0,C 180,E1 -8433.289,E2 -8433.289} C_VEL
LIN {X 0,Y 453.482,Z 288.809,A -85,B 0,C 180,E1 -8436.238,E2 -8436.238} C_VEL
LIN {X 0,Y 453.463,Z 288.809,A -85,B 0,C 180,E1 -8439.117,E2 -8439.117} C_VEL
LIN {X 0,Y 453.472,Z 288.809,A -85,B 0,C 180,E1 -8441.943,E2 -8441.943} C_VEL
LIN {X 0,Y 453.507,Z 288.806,A -85,B 0,C 180,E1 -8444.725,E2 -8444.725} C_VEL
LIN {X 0,Y 453.547,Z 288.804,A -85,B 0,C 180,E1 -8448.379,E2 -8448.379} C_VEL
LIN {X 0,Y 453.565,Z 288.795,A -85,B 0,C 180,E1 -8451.086,E2 -8451.086} C_VEL
LIN {X 0,Y 453.625,Z 288.79,A -85,B 0,C 180,E1 -8453.774,E2 -8453.774} C_VEL
LIN {X 0,Y 453.691,Z 288.78,A -85,B 0,C 180,E1 -8457.336,E2 -8457.336} C_VEL
LIN {X 0,Y 453.756,Z 288.779,A -85,B 0,C 180,E1 -8460,E2 -8460} C_VEL
LIN {X 0,Y 453.69,Z 288.78,A -85,B 0,C 180,E1 -8462.664,E2 -8462.664} C_VEL
LIN {X 0,Y 453.625,Z 288.791,A -85,B 0,C 180,E1 -8466.226,E2 -8466.226} C_VEL
LIN {X 0,Y 453.544,Z 288.798,A -85,B 0,C 180,E1 -8468.914,E2 -8468.914} C_VEL
LIN {X 0,Y 453.554,Z 288.797,A -85,B 0,C 180,E1 -8472.529,E2 -8472.529} C_VEL
LIN {X 0,Y 453.487,Z 288.806,A -85,B 0,C 180,E1 -8476.198,E2 -8476.198} C_VEL
LIN {X 0,Y 453.508,Z 288.804,A -85,B 0,C 180,E1 -8479.04,E2 -8479.04} C_VEL
LIN {X 0,Y 453.461,Z 288.811,A -85,B 0,C 180,E1 -8481.837,E2 -8481.837} C_VEL
LIN {X 0,Y 453.458,Z 288.809,A -85,B 0,C 180,E1 -8484.738,E2 -8484.738} C_VEL
LIN {X 0,Y 453.452,Z 288.81,A -85,B 0,C 180,E1 -8487.943,E2 -8487.943} C_VEL
LIN {X 0,Y 453.444,Z 288.812,A -85,B 0,C 180,E1 -8490.762,E2 -8490.762} C_VEL
LIN {X 0,Y 453.458,Z 288.809,A -85,B 0,C 180,E1 -8493.914,E2 -8493.914} C_VEL
LIN {X 0,Y 453.439,Z 288.818,A -85,B 0,C 180,E1 -8497.191,E2 -8497.191} C_VEL
LIN {X 0,Y 453.463,Z 288.81,A -85,B 0,C 180,E1 -8500.612,E2 -8500.612} C_VEL
LIN {X 0,Y 453.475,Z 288.809,A -85,B 0,C 180,E1 -8504.529,E2 -8504.529} C_VEL
LIN {X 0,Y 453.43,Z 288.812,A -85,B 0,C 180,E1 -8508.072,E2 -8508.072} C_VEL
LIN {X 0,Y 453.436,Z 288.819,A -85,B 0,C 180,E1 -8510.803,E2 -8510.803} C_VEL
LIN {X 0,Y 453.445,Z 288.81,A -85,B 0,C 180,E1 -8513.917,E2 -8513.917} C_VEL
LIN {X 0,Y 453.47,Z 288.809,A -85,B 0,C 180,E1 -8517.151,E2 -8517.151} C_VEL
LIN {X 0,Y 453.444,Z 288.814,A -85,B 0,C 180,E1 -8520.267,E2 -8520.267} C_VEL
LIN {X 0,Y 453.439,Z 288.811,A -85,B 0,C 180,E1 -8523.29,E2 -8523.29} C_VEL
LIN {X 0,Y 453.48,Z 288.799,A -85,B 0,C 180,E1 -8526.238,E2 -8526.238} C_VEL
LIN {X 0,Y 453.521,Z 288.923,A -85,B 0,C 180,E1 -8527.927,E2 -8527.927} C_VEL
LIN {X 0,Y 454.438,Z 295.656,A -85,B 0,C 180,E1 -8529.637,E2 -8529.637} C_VEL
LIN {X 0,Y 454.127,Z 305.414,A -85,B 0,C 180,E1 -8531.97,E2 -8531.97} C_VEL
LIN {X 0,Y 453.569,Z 319.076,A -85,B 0,C 180,E1 -8535.187,E2 -8535.187} C_VEL
LIN {X 0,Y 453.463,Z 323.774,A -85,B 0,C 180,E1 -8536.226,E2 -8536.226} C_VEL
LIN {X 0,Y 454.414,Z 329.735,A -85,B 0,C 180,E1 -8536.39,E2 -8536.39} C_VEL
LIN {X 0,Y 455.744,Z 340.457,A -85,B 0,C 180,E1 -8536.6,E2 -8536.6} C_VEL
LIN {X 0,Y 455.684,Z 349.261,A -85,B 0,C 180,E1 -8536.738,E2 -8536.738} C_VEL
LIN {X 0,Y 454.927,Z 355.098,A -85,B 0,C 180,E1 -8536.808,E2 -8536.808} C_VEL
LIN {X 0,Y 449.321,Z 374.074,A -85,B 0,C 180,E1 -8536.946,E2 -8536.946} C_VEL
LIN {X 0,Y 448.618,Z 379.909,A -85,B 0,C 180,E1 -8537.019,E2 -8537.019} C_VEL
LIN {X 0,Y 448.465,Z 400.938,A -85,B 0,C 180,E1 -8537.384,E2 -8537.384} C_VEL
LIN {X 0,Y 448.165,Z 412.052,A -85,B 0,C 180,E1 -8537.721,E2 -8537.721} C_VEL
LIN {X 0,Y 447.812,Z 422.76,A -85,B 0,C 180,E1 -8538.228,E2 -8538.228} C_VEL
LIN {X 0,Y 447.532,Z 431.614,A -85,B 0,C 180,E1 -8538.794,E2 -8538.794} C_VEL
LIN {X 0,Y 447.156,Z 440.034,A -85,B 0,C 180,E1 -8539.473,E2 -8539.473} C_VEL
LIN {X 0,Y 446.711,Z 447.982,A -85,B 0,C 180,E1 -8540.263,E2 -8540.263} C_VEL
LIN {X 0,Y 446.467,Z 453.692,A -85,B 0,C 180,E1 -8540.943,E2 -8540.943} C_VEL
LIN {X 0,Y 446.129,Z 460.066,A -85,B 0,C 180,E1 -8541.849,E2 -8541.849} C_VEL
LIN {X 0,Y 445.974,Z 465.365,A -85,B 0,C 180,E1 -8542.758,E2 -8542.758} C_VEL
LIN {X 0,Y 445.758,Z 469.79,A -85,B 0,C 180,E1 -8543.664,E2 -8543.664} C_VEL
LIN {X 0,Y 445.547,Z 474.994,A -85,B 0,C 180,E1 -8545.023,E2 -8545.023} C_VEL
LIN {X 0,Y 445.457,Z 477.668,A -85,B 0,C 180,E1 -8545.929,E2 -8545.929} C_VEL
LIN {X 0,Y 445.445,Z 480.596,A -85,B 0,C 180,E1 -8547.287,E2 -8547.287} C_VEL
LIN {X 0,Y 445.356,Z 481.878,A -85,B 0,C 180,E1 -8548.191,E2 -8548.191} C_VEL
LIN {X 0,Y 445.313,Z 482.689,A -85,B 0,C 180,E1 -8549.096,E2 -8549.096} C_VEL
LIN {X 0,Y 445.29,Z 482.997,A -85,B 0,C 180,E1 -8550,E2 -8550} C_VEL
LIN {X 0,Y 445.313,Z 482.722,A -85,B 0,C 180,E1 -8550.904,E2 -8550.904} C_VEL
LIN {X 0,Y 445.353,Z 481.977,A -85,B 0,C 180,E1 -8551.809,E2 -8551.809} C_VEL
LIN {X 0,Y 445.432,Z 480.763,A -85,B 0,C 180,E1 -8552.713,E2 -8552.713} C_VEL
LIN {X 0,Y 445.454,Z 477.905,A -85,B 0,C 180,E1 -8554.071,E2 -8554.071} C_VEL
LIN {X 0,Y 445.543,Z 475.305,A -85,B 0,C 180,E1 -8554.977,E2 -8554.977} C_VEL
LIN {X 0,Y 445.752,Z 470.185,A -85,B 0,C 180,E1 -8556.336,E2 -8556.336} C_VEL
LIN {X 0,Y 445.973,Z 464.677,A -85,B 0,C 180,E1 -8557.47,E2 -8557.47} C_VEL
LIN {X 0,Y 446.272,Z 457.765,A -85,B 0,C 180,E1 -8558.604,E2 -8558.604} C_VEL
LIN {X 0,Y 446.683,Z 449.828,A -85,B 0,C 180,E1 -8559.623,E2 -8559.623} C_VEL
LIN {X 0,Y 447.036,Z 442.261,A -85,B 0,C 180,E1 -8560.416,E2 -8560.416} C_VEL
LIN {X 0,Y 447.383,Z 434.334,A -85,B 0,C 180,E1 -8561.095,E2 -8561.095} C_VEL
LIN {X 0,Y 447.715,Z 426.152,A -85,B 0,C 180,E1 -8561.66,E2 -8561.66} C_VEL
LIN {X 0,Y 448.03,Z 417.871,A -85,B 0,C 180,E1 -8562.111,E2 -8562.111} C_VEL
LIN {X 0,Y 448.238,Z 408.937,A -85,B 0,C 180,E1 -8562.479,E2 -8562.479} C_VEL
LIN {X 0,Y 448.505,Z 399.218,A -85,B 0,C 180,E1 -8562.746,E2 -8562.746} C_VEL
LIN {X 0,Y 448.676,Z 338.49,A -85,B 0,C 180,E1 -8563.741,E2 -8563.741} C_VEL
LIN {X 0,Y 446.433,Z 323.925,A -85,B 0,C 180,E1 -8564.076,E2 -8564.076} C_VEL
LIN {X 0,Y 446.493,Z 321.422,A -85,B 0,C 180,E1 -8564.586,E2 -8564.586} C_VEL
LIN {X 0,Y 447.061,Z 307.756,A -85,B 0,C 180,E1 -8567.851,E2 -8567.851} C_VEL
LIN {X 0,Y 447.469,Z 297.994,A -85,B 0,C 180,E1 -8570.214,E2 -8570.214} C_VEL
LIN {X 0,Y 446.803,Z 291.433,A -85,B 0,C 180,E1 -8571.868,E2 -8571.868} C_VEL
LIN {X 0,Y 446.5,Z 289.796,A -85,B 0,C 180,E1 -8572.317,E2 -8572.317} C_VEL
LIN {X 0,Y 446.42,Z 289.691,A -85,B 0,C 180,E1 -8575.154,E2 -8575.154} C_VEL
LIN {X 0,Y 446.435,Z 289.685,A -85,B 0,C 180,E1 -8578.181,E2 -8578.181} C_VEL
LIN {X 0,Y 446.412,Z 289.691,A -85,B 0,C 180,E1 -8581.3,E2 -8581.3} C_VEL
LIN {X 0,Y 446.418,Z 289.685,A -85,B 0,C 180,E1 -8584.523,E2 -8584.523} C_VEL
LIN {X 0,Y 446.406,Z 289.687,A -85,B 0,C 180,E1 -8588.078,E2 -8588.078} C_VEL
LIN {X 0,Y 446.395,Z 289.694,A -85,B 0,C 180,E1 -8591.394,E2 -8591.394} C_VEL
LIN {X 0,Y 446.444,Z 289.69,A -85,B 0,C 180,E1 -8595.103,E2 -8595.103} C_VEL
LIN {X 0,Y 446.394,Z 289.691,A -85,B 0,C 180,E1 -8598.605,E2 -8598.605} C_VEL
LIN {X 0,Y 446.403,Z 289.687,A -85,B 0,C 180,E1 -8601.921,E2 -8601.921} C_VEL
LIN {X 0,Y 446.414,Z 289.687,A -85,B 0,C 180,E1 -8605.476,E2 -8605.476} C_VEL
LIN {X 0,Y 446.4,Z 289.694,A -85,B 0,C 180,E1 -8608.698,E2 -8608.698} C_VEL
LIN {X 0,Y 446.415,Z 289.686,A -85,B 0,C 180,E1 -8611.836,E2 -8611.836} C_VEL
LIN {X 0,Y 446.412,Z 289.691,A -85,B 0,C 180,E1 -8614.845,E2 -8614.845} C_VEL
LIN {X 0,Y 446.437,Z 289.687,A -85,B 0,C 180,E1 -8618.245,E2 -8618.245} C_VEL
LIN {X 0,Y 446.428,Z 289.684,A -85,B 0,C 180,E1 -8621.648,E2 -8621.648} C_VEL
LIN {X 0,Y 446.447,Z 289.689,A -85,B 0,C 180,E1 -8624.477,E2 -8624.477} C_VEL
LIN {X 0,Y 446.507,Z 289.674,A -85,B 0,C 180,E1 -8627.384,E2 -8627.384} C_VEL
LIN {X 0,Y 446.519,Z 289.674,A -85,B 0,C 180,E1 -8630.944,E2 -8630.944} C_VEL
LIN {X 0,Y 446.596,Z 289.665,A -85,B 0,C 180,E1 -8633.675,E2 -8633.675} C_VEL
LIN {X 0,Y 446.641,Z 289.658,A -85,B 0,C 180,E1 -8637.294,E2 -8637.294} C_VEL
LIN {X 0,Y 446.706,Z 289.657,A -85,B 0,C 180,E1 -8640,E2 -8640} C_VEL
LIN {X 0,Y 446.64,Z 289.658,A -85,B 0,C 180,E1 -8642.706,E2 -8642.706} C_VEL
LIN {X 0,Y 446.595,Z 289.666,A -85,B 0,C 180,E1 -8646.324,E2 -8646.324} C_VEL
LIN {X 0,Y 446.497,Z 289.676,A -85,B 0,C 180,E1 -8649.056,E2 -8649.056} C_VEL
LIN {X 0,Y 446.511,Z 289.674,A -85,B 0,C 180,E1 -8652.73,E2 -8652.73} C_VEL
LIN {X 0,Y 446.444,Z 289.684,A -85,B 0,C 180,E1 -8656.209,E2 -8656.209} C_VEL
LIN {X 0,Y 446.457,Z 289.685,A -85,B 0,C 180,E1 -8659.304,E2 -8659.304} C_VEL
LIN {X 0,Y 446.398,Z 289.688,A -85,B 0,C 180,E1 -8662.201,E2 -8662.201} C_VEL
LIN {X 0,Y 446.41,Z 289.691,A -85,B 0,C 180,E1 -8665.155,E2 -8665.155} C_VEL
LIN {X 0,Y 446.407,Z 289.687,A -85,B 0,C 180,E1 -8668.184,E2 -8668.184} C_VEL
LIN {X 0,Y 446.399,Z 289.695,A -85,B 0,C 180,E1 -8671.302,E2 -8671.302} C_VEL
LIN {X 0,Y 446.412,Z 289.687,A -85,B 0,C 180,E1 -8674.524,E2 -8674.524} C_VEL
LIN {X 0,Y 446.402,Z 289.687,A -85,B 0,C 180,E1 -8678.079,E2 -8678.079} C_VEL
LIN {X 0,Y 446.392,Z 289.691,A -85,B 0,C 180,E1 -8681.395,E2 -8681.395} C_VEL
LIN {X 0,Y 446.443,Z 289.687,A -85,B 0,C 180,E1 -8685.105,E2 -8685.105} C_VEL
LIN {X 0,Y 446.394,Z 289.694,A -85,B 0,C 180,E1 -8688.606,E2 -8688.606} C_VEL
LIN {X 0,Y 446.399,Z 289.688,A -85,B 0,C 180,E1 -8691.923,E2 -8691.923} C_VEL
LIN {X 0,Y 446.416,Z 289.686,A -85,B 0,C 180,E1 -8695.477,E2 -8695.477} C_VEL
LIN {X 0,Y 446.405,Z 289.693,A -85,B 0,C 180,E1 -8698.7,E2 -8698.7} C_VEL
LIN {X 0,Y 446.42,Z 289.686,A -85,B 0,C 180,E1 -8701.837,E2 -8701.837} C_VEL
LIN {X 0,Y 446.418,Z 289.691,A -85,B 0,C 180,E1 -8704.846,E2 -8704.846} C_VEL
LIN {X 0,Y 446.478,Z 289.837,A -85,B 0,C 180,E1 -8707.743,E2 -8707.743} C_VEL
LIN {X 0,Y 447.401,Z 295.86,A -85,B 0,C 180,E1 -8709.303,E2 -8709.303} C_VEL
LIN {X 0,Y 447.288,Z 303.667,A -85,B 0,C 180,E1 -8711.21,E2 -8711.21} C_VEL
LIN {X 0,Y 446.651,Z 317.33,A -85,B 0,C 180,E1 -8714.485,E2 -8714.485} C_VEL
LIN {X 0,Y 446.45,Z 323.709,A -85,B 0,C 180,E1 -8715.95,E2 -8715.95} C_VEL
LIN {X 0,Y 447.179,Z 328.548,A -85,B 0,C 180,E1 -8716.097,E2 -8716.097} C_VEL
LIN {X 0,Y 448.915,Z 340.264,A -85,B 0,C 180,E1 -8716.341,E2 -8716.341} C_VEL
LIN {X 0,Y 448.441,Z 399.743,A -85,B 0,C 180,E1 -8717.309,E2 -8717.309} C_VEL
LIN {X 0,Y 448.214,Z 409.298,A -85,B 0,C 180,E1 -8717.578,E2 -8717.578} C_VEL
LIN {X 0,Y 448.015,Z 419.342,A -85,B 0,C 180,E1 -8718.004,E2 -8718.004} C_VEL
LIN {X 0,Y 447.535,Z 430.745,A -85,B 0,C 180,E1 -8718.68,E2 -8718.68} C_VEL
LIN {X 0,Y 447.151,Z 439.32,A -85,B 0,C 180,E1 -8719.358,E2 -8719.358} C_VEL
LIN {X 0,Y 446.763,Z 447.385,A -85,B 0,C 180,E1 -8720.15,E2 -8720.15} C_VEL
LIN {X 0,Y 446.439,Z 454.046,A -85,B 0,C 180,E1 -8720.943,E2 -8720.943} C_VEL
LIN {X 0,Y 446.117,Z 460.367,A -85,B 0,C 180,E1 -8721.849,E2 -8721.849} C_VEL
LIN {X 0,Y 445.913,Z 465.618,A -85,B 0,C 180,E1 -8722.757,E2 -8722.757} C_VEL
LIN {X 0,Y 445.763,Z 469.995,A -85,B 0,C 180,E1 -8723.664,E2 -8723.664} C_VEL
LIN {X 0,Y 445.544,Z 475.155,A -85,B 0,C 180,E1 -8725.023,E2 -8725.023} C_VEL
LIN {X 0,Y 445.443,Z 478.941,A -85,B 0,C 180,E1 -8726.382,E2 -8726.382} C_VEL
LIN {X 0,Y 445.443,Z 480.682,A -85,B 0,C 180,E1 -8727.287,E2 -8727.287} C_VEL
LIN {X 0,Y 445.355,Z 481.93,A -85,B 0,C 180,E1 -8728.191,E2 -8728.191} C_VEL
LIN {X 0,Y 445.313,Z 482.706,A -85,B 0,C 180,E1 -8729.096,E2 -8729.096} C_VEL
LIN {X 0,Y 445.289,Z 483,A -85,B 0,C 180,E1 -8730,E2 -8730} C_VEL
LIN {X 0,Y 445.313,Z 482.705,A -85,B 0,C 180,E1 -8730.904,E2 -8730.904} C_VEL
LIN {X 0,Y 445.355,Z 481.926,A -85,B 0,C 180,E1 -8731.809,E2 -8731.809} C_VEL
LIN {X 0,Y 445.443,Z 480.676,A -85,B 0,C 180,E1 -8732.713,E2 -8732.713} C_VEL
LIN {X 0,Y 445.455,Z 477.782,A -85,B 0,C 180,E1 -8734.071,E2 -8734.071} C_VEL
LIN {X 0,Y 445.544,Z 475.144,A -85,B 0,C 180,E1 -8734.977,E2 -8734.977} C_VEL
LIN {X 0,Y 445.756,Z 469.98,A -85,B 0,C 180,E1 -8736.336,E2 -8736.336} C_VEL
LIN {X 0,Y 446.012,Z 463.174,A -85,B 0,C 180,E1 -8737.697,E2 -8737.697} C_VEL
LIN {X 0,Y 446.325,Z 455.729,A -85,B 0,C 180,E1 -8738.831,E2 -8738.831} C_VEL
LIN {X 0,Y 446.696,Z 448.384,A -85,B 0,C 180,E1 -8739.737,E2 -8739.737} C_VEL
LIN {X 0,Y 447.09,Z 440.517,A -85,B 0,C 180,E1 -8740.529,E2 -8740.529} C_VEL
LIN {X 0,Y 447.486,Z 432.203,A -85,B 0,C 180,E1 -8741.207,E2 -8741.207} C_VEL
LIN {X 0,Y 447.78,Z 423.494,A -85,B 0,C 180,E1 -8741.773,E2 -8741.773} C_VEL
LIN {X 0,Y 448.178,Z 411.698,A -85,B 0,C 180,E1 -8742.336,E2 -8742.336} C_VEL
LIN {X 0,Y 448.388,Z 401.671,A -85,B 0,C 180,E1 -8742.647,E2 -8742.647} C_VEL
LIN {X 0,Y 448.631,Z 379.546,A -85,B 0,C 180,E1 -8743.032,E2 -8743.032} C_VEL
LIN {X 0,Y 448.684,Z 338.445,A -85,B 0,C 180,E1 -8743.692,E2 -8743.692} C_VEL
LIN {X 0,Y 446.458,Z 323.925,A -85,B 0,C 180,E1 -8744.026,E2 -8744.026} C_VEL
LIN {X 0,Y 446.496,Z 321.218,A -85,B 0,C 180,E1 -8744.586,E2 -8744.586} C_VEL
LIN {X 0,Y 447.059,Z 307.553,A -85,B 0,C 180,E1 -8747.851,E2 -8747.851} C_VEL
LIN {X 0,Y 447.461,Z 297.792,A -85,B 0,C 180,E1 -8750.214,E2 -8750.214} C_VEL
LIN {X 0,Y 446.757,Z 291.297,A -85,B 0,C 180,E1 -8751.854,E2 -8751.854} C_VEL
LIN {X 0,Y 446.476,Z 289.755,A -85,B 0,C 180,E1 -8752.318,E2 -8752.318} C_VEL
LIN {X 0,Y 446.418,Z 289.691,A -85,B 0,C 180,E1 -8755.154,E2 -8755.154} C_VEL
LIN {X 0,Y 446.433,Z 289.684,A -85,B 0,C 180,E1 -8758.181,E2 -8758.181} C_VEL
LIN {X 0,Y 446.405,Z 289.693,A -85,B 0,C 180,E1 -8761.3,E2 -8761.3} C_VEL
LIN {X 0,Y 446.416,Z 289.686,A -85,B 0,C 180,E1 -8764.523,E2 -8764.523} C_VEL
LIN {X 0,Y 446.405,Z 289.687,A -85,B 0,C 180,E1 -8768.078,E2 -8768.078} C_VEL
LIN {X 0,Y 446.394,Z 289.694,A -85,B 0,C 180,E1 -8771.394,E2 -8771.394} C_VEL
LIN {X 0,Y 446.443,Z 289.69,A -85,B 0,C 180,E1 -8775.104,E2 -8775.104} C_VEL
LIN {X 0,Y 446.393,Z 289.691,A -85,B 0,C 180,E1 -8778.605,E2 -8778.605} C_VEL
LIN {X 0,Y 446.402,Z 289.687,A -85,B 0,C 180,E1 -8781.921,E2 -8781.921} C_VEL
LIN {X 0,Y 446.412,Z 289.687,A -85,B 0,C 180,E1 -8785.476,E2 -8785.476} C_VEL
LIN {X 0,Y 446.399,Z 289.694,A -85,B 0,C 180,E1 -8788.698,E2 -8788.698} C_VEL
LIN {X 0,Y 446.415,Z 289.686,A -85,B 0,C 180,E1 -8791.836,E2 -8791.836} C_VEL
LIN {X 0,Y 446.411,Z 289.691,A -85,B 0,C 180,E1 -8794.845,E2 -8794.845} C_VEL
LIN {X 0,Y 446.437,Z 289.687,A -85,B 0,C 180,E1 -8798.246,E2 -8798.246} C_VEL
LIN {X 0,Y 446.427,Z 289.684,A -85,B 0,C 180,E1 -8801.648,E2 -8801.648} C_VEL
LIN {X 0,Y 446.447,Z 289.689,A -85,B 0,C 180,E1 -8804.478,E2 -8804.478} C_VEL
LIN {X 0,Y 446.506,Z 289.674,A -85,B 0,C 180,E1 -8807.384,E2 -8807.384} C_VEL
LIN {X 0,Y 446.514,Z 289.674,A -85,B 0,C 180,E1 -8810.944,E2 -8810.944} C_VEL
LIN {X 0,Y 446.595,Z 289.665,A -85,B 0,C 180,E1 -8813.676,E2 -8813.676} C_VEL
LIN {X 0,Y 446.641,Z 289.658,A -85,B 0,C 180,E1 -8817.294,E2 -8817.294} C_VEL
LIN {X 0,Y 446.706,Z 289.657,A -85,B 0,C 180,E1 -8820,E2 -8820} C_VEL
LIN {X 0,Y 446.64,Z 289.658,A -85,B 0,C 180,E1 -8822.706,E2 -8822.706} C_VEL
LIN {X 0,Y 446.595,Z 289.666,A -85,B 0,C 180,E1 -8826.325,E2 -8826.325} C_VEL
LIN {X 0,Y 446.495,Z 289.676,A -85,B 0,C 180,E1 -8829.056,E2 -8829.056} C_VEL
LIN {X 0,Y 446.511,Z 289.674,A -85,B 0,C 180,E1 -8832.73,E2 -8832.73} C_VEL
LIN {X 0,Y 446.44,Z 289.684,A -85,B 0,C 180,E1 -8836.207,E2 -8836.207} C_VEL
LIN {X 0,Y 446.457,Z 289.685,A -85,B 0,C 180,E1 -8839.304,E2 -8839.304} C_VEL
LIN {X 0,Y 446.399,Z 289.688,A -85,B 0,C 180,E1 -8842.201,E2 -8842.201} C_VEL
LIN {X 0,Y 446.411,Z 289.691,A -85,B 0,C 180,E1 -8845.155,E2 -8845.155} C_VEL
LIN {X 0,Y 446.408,Z 289.687,A -85,B 0,C 180,E1 -8848.184,E2 -8848.184} C_VEL
LIN {X 0,Y 446.385,Z 289.697,A -85,B 0,C 180,E1 -8851.303,E2 -8851.303} C_VEL
LIN {X 0,Y 446.413,Z 289.687,A -85,B 0,C 180,E1 -8854.525,E2 -8854.525} C_VEL
LIN {X 0,Y 446.397,Z 289.688,A -85,B 0,C 180,E1 -8858.078,E2 -8858.078} C_VEL
LIN {X 0,Y 446.393,Z 289.692,A -85,B 0,C 180,E1 -8861.395,E2 -8861.395} C_VEL
LIN {X 0,Y 446.444,Z 289.688,A -85,B 0,C 180,E1 -8865.105,E2 -8865.105} C_VEL
LIN {X 0,Y 446.395,Z 289.693,A -85,B 0,C 180,E1 -8868.606,E2 -8868.606} C_VEL
LIN {X 0,Y 446.4,Z 289.688,A -85,B 0,C 180,E1 -8871.924,E2 -8871.924} C_VEL
LIN {X 0,Y 446.418,Z 289.686,A -85,B 0,C 180,E1 -8875.477,E2 -8875.477} C_VEL
LIN {X 0,Y 446.389,Z 289.695,A -85,B 0,C 180,E1 -8878.698,E2 -8878.698} C_VEL
LIN {X 0,Y 446.4,Z 289.688,A -85,B 0,C 180,E1 -8881.842,E2 -8881.842} C_VEL
LIN {X 0,Y 446.419,Z 289.691,A -85,B 0,C 180,E1 -8884.846,E2 -8884.846} C_VEL
LIN {X 0,Y 446.5,Z 289.866,A -85,B 0,C 180,E1 -8887.805,E2 -8887.805} C_VEL
LIN {X 0,Y 447.36,Z 295.658,A -85,B 0,C 180,E1 -8889.301,E2 -8889.301} C_VEL
LIN {X 0,Y 447.29,Z 303.465,A -85,B 0,C 180,E1 -8891.21,E2 -8891.21} C_VEL
LIN {X 0,Y 446.653,Z 317.126,A -85,B 0,C 180,E1 -8894.485,E2 -8894.485} C_VEL
LIN {X 0,Y 446.451,Z 323.777,A -85,B 0,C 180,E1 -8896.006,E2 -8896.006} C_VEL
LIN {X 0,Y 447.485,Z 330.34,A -85,B 0,C 180,E1 -8896.184,E2 -8896.184} C_VEL
LIN {X 0,Y 448.833,Z 340.328,A -85,B 0,C 180,E1 -8896.388,E2 -8896.388} C_VEL
LIN {X 0,Y 448.618,Z 379.909,A -85,B 0,C 180,E1 -8897.019,E2 -8897.019} C_VEL
LIN {X 0,Y 447.859,Z 385.76,A -85,B 0,C 180,E1 -8897.086,E2 -8897.086} C_VEL
LIN {X 0,Y 442.156,Z 403.693,A -85,B 0,C 180,E1 -8897.264,E2 -8897.264} C_VEL
LIN {X 0,Y 441.384,Z 408.451,A -85,B 0,C 180,E1 -8897.401,E2 -8897.401} C_VEL
LIN {X 0,Y 441.309,Z 410.358,A -85,B 0,C 180,E1 -8897.467,E2 -8897.467} C_VEL
LIN {X 0,Y 440.948,Z 421.812,A -85,B 0,C 180,E1 -8897.984,E2 -8897.984} C_VEL
LIN {X 0,Y 440.579,Z 431.62,A -85,B 0,C 180,E1 -8898.615,E2 -8898.615} C_VEL
LIN {X 0,Y 440.165,Z 440.039,A -85,B 0,C 180,E1 -8899.303,E2 -8899.303} C_VEL
LIN {X 0,Y 439.713,Z 447.986,A -85,B 0,C 180,E1 -8900.107,E2 -8900.107} C_VEL
LIN {X 0,Y 439.44,Z 453.695,A -85,B 0,C 180,E1 -8900.797,E2 -8900.797} C_VEL
LIN {X 0,Y 439.1,Z 460.068,A -85,B 0,C 180,E1 -8901.718,E2 -8901.718} C_VEL
LIN {X 0,Y 438.846,Z 466.541,A -85,B 0,C 180,E1 -8902.871,E2 -8902.871} C_VEL
LIN {X 0,Y 438.642,Z 471.705,A -85,B 0,C 180,E1 -8904.022,E2 -8904.022} C_VEL
LIN {X 0,Y 438.399,Z 476.488,A -85,B 0,C 180,E1 -8905.403,E2 -8905.403} C_VEL
LIN {X 0,Y 438.347,Z 478.82,A -85,B 0,C 180,E1 -8906.323,E2 -8906.323} C_VEL
LIN {X 0,Y 438.355,Z 480.597,A -85,B 0,C 180,E1 -8907.243,E2 -8907.243} C_VEL
LIN {X 0,Y 438.279,Z 481.878,A -85,B 0,C 180,E1 -8908.162,E2 -8908.162} C_VEL
LIN {X 0,Y 438.228,Z 482.689,A -85,B 0,C 180,E1 -8909.081,E2 -8909.081} C_VEL
LIN {X 0,Y 438.204,Z 482.997,A -85,B 0,C 180,E1 -8910,E2 -8910} C_VEL
LIN {X 0,Y 438.229,Z 482.722,A -85,B 0,C 180,E1 -8910.919,E2 -8910.919} C_VEL
LIN {X 0,Y 438.275,Z 481.977,A -85,B 0,C 180,E1 -8911.838,E2 -8911.838} C_VEL
LIN {X 0,Y 438.344,Z 480.762,A -85,B 0,C 180,E1 -8912.757,E2 -8912.757} C_VEL
LIN {X 0,Y 438.362,Z 477.904,A -85,B 0,C 180,E1 -8914.137,E2 -8914.137} C_VEL
LIN {X 0,Y 438.482,Z 475.304,A -85,B 0,C 180,E1 -8915.057,E2 -8915.057} C_VEL
LIN {X 0,Y 438.681,Z 470.183,A -85,B 0,C 180,E1 -8916.439,E2 -8916.439} C_VEL
LIN {X 0,Y 438.915,Z 464.675,A -85,B 0,C 180,E1 -8917.591,E2 -8917.591} C_VEL
LIN {X 0,Y 439.233,Z 457.762,A -85,B 0,C 180,E1 -8918.743,E2 -8918.743} C_VEL
LIN {X 0,Y 439.655,Z 449.824,A -85,B 0,C 180,E1 -8919.778,E2 -8919.778} C_VEL
LIN {X 0,Y 440.049,Z 442.256,A -85,B 0,C 180,E1 -8920.583,E2 -8920.583} C_VEL
LIN {X 0,Y 440.429,Z 434.328,A -85,B 0,C 180,E1 -8921.272,E2 -8921.272} C_VEL
LIN {X 0,Y 440.749,Z 426.145,A -85,B 0,C 180,E1 -8921.847,E2 -8921.847} C_VEL
LIN {X 0,Y 441.101,Z 417.861,A -85,B 0,C 180,E1 -8922.304,E2 -8922.304} C_VEL
LIN {X 0,Y 441.327,Z 408.924,A -85,B 0,C 180,E1 -8922.677,E2 -8922.677} C_VEL
LIN {X 0,Y 441.58,Z 399.346,A -85,B 0,C 180,E1 -8922.946,E2 -8922.946} C_VEL
LIN {X 0,Y 441.824,Z 339.419,A -85,B 0,C 180,E1 -8923.942,E2 -8923.942} C_VEL
LIN {X 0,Y 439.455,Z 324.157,A -85,B 0,C 180,E1 -8924.293,E2 -8924.293} C_VEL
LIN {X 0,Y 439.422,Z 323.504,A -85,B 0,C 180,E1 -8924.353,E2 -8924.353} C_VEL
LIN {X 0,Y 439.922,Z 311.659,A -85,B 0,C 180,E1 -8927.19,E2 -8927.19} C_VEL
LIN {X 0,Y 440.463,Z 299.947,A -85,B 0,C 180,E1 -8930.062,E2 -8930.062} C_VEL
LIN {X 0,Y 440.036,Z 294.087,A -85,B 0,C 180,E1 -8931.551,E2 -8931.551} C_VEL
LIN {X 0,Y 439.454,Z 290.646,A -85,B 0,C 180,E1 -8932.489,E2 -8932.489} C_VEL
LIN {X 0,Y 439.365,Z 290.572,A -85,B 0,C 180,E1 -8935.587,E2 -8935.587} C_VEL
LIN {X 0,Y 439.388,Z 290.561,A -85,B 0,C 180,E1 -8938.675,E2 -8938.675} C_VEL
LIN {X 0,Y 439.363,Z 290.566,A -85,B 0,C 180,E1 -8942.029,E2 -8942.029} C_VEL
LIN {X 0,Y 439.387,Z 290.568,A -85,B 0,C 180,E1 -8945.339,E2 -8945.339} C_VEL
LIN {X 0,Y 439.358,Z 290.566,A -85,B 0,C 180,E1 -8948.596,E2 -8948.596} C_VEL
LIN {X 0,Y 439.343,Z 290.567,A -85,B 0,C 180,E1 -8952.209,E2 -8952.209} C_VEL
LIN {X 0,Y 439.391,Z 290.567,A -85,B 0,C 180,E1 -8955.269,E2 -8955.269} C_VEL
LIN {X 0,Y 439.348,Z 290.574,A -85,B 0,C 180,E1 -8959.015,E2 -8959.015} C_VEL
LIN {X 0,Y 439.36,Z 290.566,A -85,B 0,C 180,E1 -8961.608,E2 -8961.608} C_VEL
LIN {X 0,Y 439.387,Z 290.568,A -85,B 0,C 180,E1 -8964.843,E2 -8964.843} C_VEL
LIN {X 0,Y 439.358,Z 290.566,A -85,B 0,C 180,E1 -8968.138,E2 -8968.138} C_VEL
LIN {X 0,Y 439.379,Z 290.562,A -85,B 0,C 180,E1 -8971.609,E2 -8971.609} C_VEL
LIN {X 0,Y 439.357,Z 290.569,A -85,B 0,C 180,E1 -8974.412,E2 -8974.412} C_VEL
LIN {X 0,Y 439.351,Z 290.566,A -85,B 0,C 180,E1 -8977.424,E2 -8977.424} C_VEL
LIN {X 0,Y 439.431,Z 290.561,A -85,B 0,C 180,E1 -8980.663,E2 -8980.663} C_VEL
LIN {X 0,Y 439.406,Z 290.564,A -85,B 0,C 180,E1 -8984.222,E2 -8984.222} C_VEL
LIN {X 0,Y 439.475,Z 290.55,A -85,B 0,C 180,E1 -8987.285,E2 -8987.285} C_VEL
LIN {X 0,Y 439.483,Z 290.551,A -85,B 0,C 180,E1 -8990.798,E2 -8990.798} C_VEL
LIN {X 0,Y 439.549,Z 290.542,A -85,B 0,C 180,E1 -8993.574,E2 -8993.574} C_VEL
LIN {X 0,Y 439.394,Z 290.561,A -85,B 0,C 180,E1 -8995.413,E2 -8995.413} C_VEL
LIN {X 0,Y 439.615,Z 290.539,A -85,B 0,C 180,E1 -8998.168,E2 -8998.168} C_VEL
LIN {X 0,Y 439.657,Z 290.535,A -85,B 0,C 180,E1 -9000,E2 -9000} C_VEL
LIN {X 0,Y 439.591,Z 290.536,A -85,B 0,C 180,E1 -9002.749,E2 -9002.749} C_VEL
LIN {X 0,Y 439.548,Z 290.543,A -85,B 0,C 180,E1 -9006.426,E2 -9006.426} C_VEL
LIN {X 0,Y 439.463,Z 290.553,A -85,B 0,C 180,E1 -9009.202,E2 -9009.202} C_VEL
LIN {X 0,Y 439.455,Z 290.553,A -85,B 0,C 180,E1 -9012.938,E2 -9012.938} C_VEL
LIN {X 0,Y 439.392,Z 290.561,A -85,B 0,C 180,E1 -9016.328,E2 -9016.328} C_VEL
LIN {X 0,Y 439.389,Z 290.568,A -85,B 0,C 180,E1 -9019.627,E2 -9019.627} C_VEL
LIN {X 0,Y 439.343,Z 290.567,A -85,B 0,C 180,E1 -9022.576,E2 -9022.576} C_VEL
LIN {X 0,Y 439.356,Z 290.57,A -85,B 0,C 180,E1 -9025.588,E2 -9025.588} C_VEL
LIN {X 0,Y 439.372,Z 290.564,A -85,B 0,C 180,E1 -9028.677,E2 -9028.677} C_VEL
LIN {X 0,Y 439.354,Z 290.566,A -85,B 0,C 180,E1 -9032.029,E2 -9032.029} C_VEL
LIN {X 0,Y 439.382,Z 290.567,A -85,B 0,C 180,E1 -9035.34,E2 -9035.34} C_VEL
LIN {X 0,Y 439.354,Z 290.568,A -85,B 0,C 180,E1 -9038.598,E2 -9038.598} C_VEL
LIN {X 0,Y 439.341,Z 290.567,A -85,B 0,C 180,E1 -9042.211,E2 -9042.211} C_VEL
LIN {X 0,Y 439.39,Z 290.564,A -85,B 0,C 180,E1 -9045.271,E2 -9045.271} C_VEL
LIN {X 0,Y 439.348,Z 290.571,A -85,B 0,C 180,E1 -9049.017,E2 -9049.017} C_VEL
LIN {X 0,Y 439.336,Z 290.573,A -85,B 0,C 180,E1 -9052.565,E2 -9052.565} C_VEL
LIN {X 0,Y 439.389,Z 290.566,A -85,B 0,C 180,E1 -9054.844,E2 -9054.844} C_VEL
LIN {X 0,Y 439.365,Z 290.567,A -85,B 0,C 180,E1 -9058.14,E2 -9058.14} C_VEL
LIN {X 0,Y 439.383,Z 290.562,A -85,B 0,C 180,E1 -9061.61,E2 -9061.61} C_VEL
LIN {X 0,Y 439.364,Z 290.572,A -85,B 0,C 180,E1 -9064.413,E2 -9064.413} C_VEL
LIN {X 0,Y 439.45,Z 290.729,A -85,B 0,C 180,E1 -9067.596,E2 -9067.596} C_VEL
LIN {X 0,Y 440.303,Z 295.862,A -85,B 0,C 180,E1 -9068.953,E2 -9068.953} C_VEL
LIN {X 0,Y 440.402,Z 301.717,A -85,B 0,C 180,E1 -9070.421,E2 -9070.421} C_VEL
LIN {X 0,Y 439.745,Z 315.83,A -85,B 0,C 180,E1 -9073.869,E2 -9073.869} C_VEL
LIN {X 0,Y 439.41,Z 323.592,A -85,B 0,C 180,E1 -9075.706,E2 -9075.706} C_VEL
LIN {X 0,Y 439.793,Z 326.358,A -85,B 0,C 180,E1 -9075.822,E2 -9075.822} C_VEL
LIN {X 0,Y 442.01,Z 340.536,A -85,B 0,C 180,E1 -9076.127,E2 -9076.127} C_VEL
LIN {X 0,Y 441.535,Z 399.79,A -85,B 0,C 180,E1 -9077.107,E2 -9077.107} C_VEL
LIN {X 0,Y 441.292,Z 409.307,A -85,B 0,C 180,E1 -9077.38,E2 -9077.38} C_VEL
LIN {X 0,Y 441.067,Z 419.348,A -85,B 0,C 180,E1 -9077.812,E2 -9077.812} C_VEL
LIN {X 0,Y 440.578,Z 430.748,A -85,B 0,C 180,E1 -9078.499,E2 -9078.499} C_VEL
LIN {X 0,Y 440.18,Z 439.323,A -85,B 0,C 180,E1 -9079.187,E2 -9079.187} C_VEL
LIN {X 0,Y 439.773,Z 447.388,A -85,B 0,C 180,E1 -9079.992,E2 -9079.992} C_VEL
LIN {X 0,Y 439.41,Z 454.048,A -85,B 0,C 180,E1 -9080.797,E2 -9080.797} C_VEL
LIN {X 0,Y 439.091,Z 460.369,A -85,B 0,C 180,E1 -9081.718,E2 -9081.718} C_VEL
LIN {X 0,Y 438.872,Z 465.619,A -85,B 0,C 180,E1 -9082.64,E2 -9082.64} C_VEL
LIN {X 0,Y 438.691,Z 469.996,A -85,B 0,C 180,E1 -9083.561,E2 -9083.561} C_VEL
LIN {X 0,Y 438.483,Z 475.155,A -85,B 0,C 180,E1 -9084.943,E2 -9084.943} C_VEL
LIN {X 0,Y 438.346,Z 478.942,A -85,B 0,C 180,E1 -9086.323,E2 -9086.323} C_VEL
LIN {X 0,Y 438.354,Z 480.683,A -85,B 0,C 180,E1 -9087.243,E2 -9087.243} C_VEL
LIN {X 0,Y 438.278,Z 481.93,A -85,B 0,C 180,E1 -9088.162,E2 -9088.162} C_VEL
LIN {X 0,Y 438.228,Z 482.706,A -85,B 0,C 180,E1 -9089.081,E2 -9089.081} C_VEL
LIN {X 0,Y 438.203,Z 483,A -85,B 0,C 180,E1 -9090,E2 -9090} C_VEL
LIN {X 0,Y 438.228,Z 482.705,A -85,B 0,C 180,E1 -9090.919,E2 -9090.919} C_VEL
LIN {X 0,Y 438.278,Z 481.926,A -85,B 0,C 180,E1 -9091.838,E2 -9091.838} C_VEL
LIN {X 0,Y 438.354,Z 480.676,A -85,B 0,C 180,E1 -9092.757,E2 -9092.757} C_VEL
LIN {X 0,Y 438.363,Z 477.782,A -85,B 0,C 180,E1 -9094.137,E2 -9094.137} C_VEL
LIN {X 0,Y 438.483,Z 475.144,A -85,B 0,C 180,E1 -9095.057,E2 -9095.057} C_VEL
LIN {X 0,Y 438.68,Z 469.979,A -85,B 0,C 180,E1 -9096.439,E2 -9096.439} C_VEL
LIN {X 0,Y 438.952,Z 463.172,A -85,B 0,C 180,E1 -9097.822,E2 -9097.822} C_VEL
LIN {X 0,Y 439.311,Z 455.727,A -85,B 0,C 180,E1 -9098.973,E2 -9098.973} C_VEL
LIN {X 0,Y 439.698,Z 448.382,A -85,B 0,C 180,E1 -9099.894,E2 -9099.894} C_VEL
LIN {X 0,Y 440.107,Z 440.514,A -85,B 0,C 180,E1 -9100.698,E2 -9100.698} C_VEL
LIN {X 0,Y 440.524,Z 432.199,A -85,B 0,C 180,E1 -9101.386,E2 -9101.386} C_VEL
LIN {X 0,Y 440.955,Z 421.579,A -85,B 0,C 180,E1 -9102.074,E2 -9102.074} C_VEL
LIN {X 0,Y 441.283,Z 410.026,A -85,B 0,C 180,E1 -9102.591,E2 -9102.591} C_VEL
LIN {X 0,Y 441.525,Z 400.361,A -85,B 0,C 180,E1 -9102.876,E2 -9102.876} C_VEL
LIN {X 0,Y 441.863,Z 339.708,A -85,B 0,C 180,E1 -9103.887,E2 -9103.887} C_VEL
LIN {X 0,Y 439.452,Z 324.048,A -85,B 0,C 180,E1 -9104.245,E2 -9104.245} C_VEL
LIN {X 0,Y 439.44,Z 322.29,A -85,B 0,C 180,E1 -9104.565,E2 -9104.565} C_VEL
LIN {X 0,Y 439.982,Z 309.504,A -85,B 0,C 180,E1 -9107.667,E2 -9107.667} C_VEL
LIN {X 0,Y 440.458,Z 299.745,A -85,B 0,C 180,E1 -9110.062,E2 -9110.062} C_VEL
LIN {X 0,Y 440.01,Z 293.886,A -85,B 0,C 180,E1 -9111.553,E2 -9111.553} C_VEL
LIN {X 0,Y 439.444,Z 290.646,A -85,B 0,C 180,E1 -9112.445,E2 -9112.445} C_VEL
LIN {X 0,Y 439.364,Z 290.572,A -85,B 0,C 180,E1 -9115.587,E2 -9115.587} C_VEL
LIN {X 0,Y 439.386,Z 290.562,A -85,B 0,C 180,E1 -9118.675,E2 -9118.675} C_VEL
LIN {X 0,Y 439.361,Z 290.566,A -85,B 0,C 180,E1 -9122.029,E2 -9122.029} C_VEL
LIN {X 0,Y 439.385,Z 290.569,A -85,B 0,C 180,E1 -9125.339,E2 -9125.339} C_VEL
LIN {X 0,Y 439.357,Z 290.566,A -85,B 0,C 180,E1 -9128.597,E2 -9128.597} C_VEL
LIN {X 0,Y 439.342,Z 290.567,A -85,B 0,C 180,E1 -9132.209,E2 -9132.209} C_VEL
LIN {X 0,Y 439.39,Z 290.567,A -85,B 0,C 180,E1 -9135.269,E2 -9135.269} C_VEL
LIN {X 0,Y 439.346,Z 290.574,A -85,B 0,C 180,E1 -9139.016,E2 -9139.016} C_VEL
LIN {X 0,Y 439.336,Z 290.571,A -85,B 0,C 180,E1 -9142.564,E2 -9142.564} C_VEL
LIN {X 0,Y 439.386,Z 290.569,A -85,B 0,C 180,E1 -9144.843,E2 -9144.843} C_VEL
LIN {X 0,Y 439.357,Z 290.566,A -85,B 0,C 180,E1 -9148.138,E2 -9148.138} C_VEL
LIN {X 0,Y 439.378,Z 290.563,A -85,B 0,C 180,E1 -9151.609,E2 -9151.609} C_VEL
LIN {X 0,Y 439.357,Z 290.57,A -85,B 0,C 180,E1 -9154.412,E2 -9154.412} C_VEL
LIN {X 0,Y 439.35,Z 290.566,A -85,B 0,C 180,E1 -9157.424,E2 -9157.424} C_VEL
LIN {X 0,Y 439.431,Z 290.561,A -85,B 0,C 180,E1 -9160.663,E2 -9160.663} C_VEL
LIN {X 0,Y 439.406,Z 290.564,A -85,B 0,C 180,E1 -9164.223,E2 -9164.223} C_VEL
LIN {X 0,Y 439.475,Z 290.55,A -85,B 0,C 180,E1 -9167.285,E2 -9167.285} C_VEL
LIN {X 0,Y 439.478,Z 290.551,A -85,B 0,C 180,E1 -9170.798,E2 -9170.798} C_VEL
LIN {X 0,Y 439.548,Z 290.542,A -85,B 0,C 180,E1 -9173.574,E2 -9173.574} C_VEL
LIN {X 0,Y 439.394,Z 290.561,A -85,B 0,C 180,E1 -9175.413,E2 -9175.413} C_VEL
LIN {X 0,Y 439.615,Z 290.539,A -85,B 0,C 180,E1 -9178.168,E2 -9178.168} C_VEL
LIN {X 0,Y 439.657,Z 290.535,A -85,B 0,C 180,E1 -9180,E2 -9180} C_VEL
LIN {X 0,Y 439.591,Z 290.536,A -85,B 0,C 180,E1 -9182.749,E2 -9182.749} C_VEL
LIN {X 0,Y 439.548,Z 290.543,A -85,B 0,C 180,E1 -9186.426,E2 -9186.426} C_VEL
LIN {X 0,Y 439.461,Z 290.553,A -85,B 0,C 180,E1 -9189.203,E2 -9189.203} C_VEL
LIN {X 0,Y 439.455,Z 290.553,A -85,B 0,C 180,E1 -9192.938,E2 -9192.938} C_VEL
LIN {X 0,Y 439.387,Z 290.562,A -85,B 0,C 180,E1 -9196.326,E2 -9196.326} C_VEL
LIN {X 0,Y 439.389,Z 290.568,A -85,B 0,C 180,E1 -9199.627,E2 -9199.627} C_VEL
LIN {X 0,Y 439.344,Z 290.567,A -85,B 0,C 180,E1 -9202.577,E2 -9202.577} C_VEL
LIN {X 0,Y 439.357,Z 290.57,A -85,B 0,C 180,E1 -9205.588,E2 -9205.588} C_VEL
LIN {X 0,Y 439.371,Z 290.564,A -85,B 0,C 180,E1 -9208.677,E2 -9208.677} C_VEL
LIN {X 0,Y 439.344,Z 290.567,A -85,B 0,C 180,E1 -9212.027,E2 -9212.027} C_VEL
LIN {X 0,Y 439.382,Z 290.567,A -85,B 0,C 180,E1 -9215.34,E2 -9215.34} C_VEL
LIN {X 0,Y 439.35,Z 290.568,A -85,B 0,C 180,E1 -9218.599,E2 -9218.599} C_VEL
LIN {X 0,Y 439.342,Z 290.567,A -85,B 0,C 180,E1 -9222.211,E2 -9222.211} C_VEL
LIN {X 0,Y 439.391,Z 290.564,A -85,B 0,C 180,E1 -9225.271,E2 -9225.271} C_VEL
LIN {X 0,Y 439.349,Z 290.571,A -85,B 0,C 180,E1 -9229.017,E2 -9229.017} C_VEL
LIN {X 0,Y 439.337,Z 290.573,A -85,B 0,C 180,E1 -9232.565,E2 -9232.565} C_VEL
LIN {X 0,Y 439.391,Z 290.566,A -85,B 0,C 180,E1 -9234.844,E2 -9234.844} C_VEL
LIN {X 0,Y 439.352,Z 290.568,A -85,B 0,C 180,E1 -9238.139,E2 -9238.139} C_VEL
LIN {X 0,Y 439.383,Z 290.562,A -85,B 0,C 180,E1 -9241.611,E2 -9241.611} C_VEL
LIN {X 0,Y 439.365,Z 290.571,A -85,B 0,C 180,E1 -9244.413,E2 -9244.413} C_VEL
LIN {X 0,Y 439.443,Z 290.719,A -85,B 0,C 180,E1 -9247.642,E2 -9247.642} C_VEL
LIN {X 0,Y 440.396,Z 297.612,A -85,B 0,C 180,E1 -9249.447,E2 -9249.447} C_VEL
LIN {X 0,Y 440.206,Z 305.418,A -85,B 0,C 180,E1 -9251.38,E2 -9251.38} C_VEL
LIN {X 0,Y 439.588,Z 319.08,A -85,B 0,C 180,E1 -9254.705,E2 -9254.705} C_VEL
LIN {X 0,Y 439.428,Z 323.757,A -85,B 0,C 180,E1 -9255.774,E2 -9255.774} C_VEL
LIN {X 0,Y 440.297,Z 329.402,A -85,B 0,C 180,E1 -9255.938,E2 -9255.938} C_VEL
LIN {X 0,Y 441.948,Z 340.674,A -85,B 0,C 180,E1 -9256.177,E2 -9256.177} C_VEL
LIN {X 0,Y 441.601,Z 399.661,A -85,B 0,C 180,E1 -9257.156,E2 -9257.156} C_VEL
LIN {X 0,Y 441.342,Z 408.745,A -85,B 0,C 180,E1 -9257.411,E2 -9257.411} C_VEL
LIN {X 0,Y 441.309,Z 410.358,A -85,B 0,C 180,E1 -9257.467,E2 -9257.467} C_VEL
LIN {X 0,Y 440.551,Z 416.015,A -85,B 0,C 180,E1 -9257.67,E2 -9257.67} C_VEL
LIN {X 0,Y 437.42,Z 424.974,A -85,B 0,C 180,E1 -9258.054,E2 -9258.054} C_VEL
LIN {X 0,Y 434.194,Z 433.484,A -85,B 0,C 180,E1 -9258.57,E2 -9258.57} C_VEL
LIN {X 0,Y 433.291,Z 438.431,A -85,B 0,C 180,E1 -9258.977,E2 -9258.977} C_VEL
LIN {X 0,Y 432.815,Z 446.969,A -85,B 0,C 180,E1 -9259.829,E2 -9259.829} C_VEL
LIN {X 0,Y 432.421,Z 453.699,A -85,B 0,C 180,E1 -9260.647,E2 -9260.647} C_VEL
LIN {X 0,Y 432.062,Z 460.071,A -85,B 0,C 180,E1 -9261.582,E2 -9261.582} C_VEL
LIN {X 0,Y 431.795,Z 466.543,A -85,B 0,C 180,E1 -9262.754,E2 -9262.754} C_VEL
LIN {X 0,Y 431.556,Z 471.707,A -85,B 0,C 180,E1 -9263.924,E2 -9263.924} C_VEL
LIN {X 0,Y 431.332,Z 476.489,A -85,B 0,C 180,E1 -9265.327,E2 -9265.327} C_VEL
LIN {X 0,Y 431.252,Z 478.821,A -85,B 0,C 180,E1 -9266.263,E2 -9266.263} C_VEL
LIN {X 0,Y 431.253,Z 480.597,A -85,B 0,C 180,E1 -9267.198,E2 -9267.198} C_VEL
LIN {X 0,Y 431.204,Z 481.879,A -85,B 0,C 180,E1 -9268.132,E2 -9268.132} C_VEL
LIN {X 0,Y 431.147,Z 482.689,A -85,B 0,C 180,E1 -9269.066,E2 -9269.066} C_VEL
LIN {X 0,Y 431.121,Z 482.997,A -85,B 0,C 180,E1 -9270,E2 -9270} C_VEL
LIN {X 0,Y 431.147,Z 482.722,A -85,B 0,C 180,E1 -9270.934,E2 -9270.934} C_VEL
LIN {X 0,Y 431.2,Z 481.976,A -85,B 0,C 180,E1 -9271.868,E2 -9271.868} C_VEL
LIN {X 0,Y 431.243,Z 480.761,A -85,B 0,C 180,E1 -9272.802,E2 -9272.802} C_VEL
LIN {X 0,Y 431.277,Z 477.903,A -85,B 0,C 180,E1 -9274.205,E2 -9274.205} C_VEL
LIN {X 0,Y 431.421,Z 475.302,A -85,B 0,C 180,E1 -9275.14,E2 -9275.14} C_VEL
LIN {X 0,Y 431.63,Z 470.181,A -85,B 0,C 180,E1 -9276.544,E2 -9276.544} C_VEL
LIN {X 0,Y 431.853,Z 464.673,A -85,B 0,C 180,E1 -9277.716,E2 -9277.716} C_VEL
LIN {X 0,Y 432.218,Z 457.758,A -85,B 0,C 180,E1 -9278.886,E2 -9278.886} C_VEL
LIN {X 0,Y 432.636,Z 449.82,A -85,B 0,C 180,E1 -9279.939,E2 -9279.939} C_VEL
LIN {X 0,Y 433.058,Z 442.252,A -85,B 0,C 180,E1 -9280.756,E2 -9280.756} C_VEL
LIN {X 0,Y 433.481,Z 434.323,A -85,B 0,C 180,E1 -9281.455,E2 -9281.455} C_VEL
LIN {X 0,Y 433.808,Z 426.138,A -85,B 0,C 180,E1 -9282.039,E2 -9282.039} C_VEL
LIN {X 0,Y 434.183,Z 417.852,A -85,B 0,C 180,E1 -9282.503,E2 -9282.503} C_VEL
LIN {X 0,Y 434.422,Z 408.911,A -85,B 0,C 180,E1 -9282.882,E2 -9282.882} C_VEL
LIN {X 0,Y 434.673,Z 399.457,A -85,B 0,C 180,E1 -9283.153,E2 -9283.153} C_VEL
LIN {X 0,Y 434.904,Z 339.627,A -85,B 0,C 180,E1 -9284.165,E2 -9284.165} C_VEL
LIN {X 0,Y 432.45,Z 324.148,A -85,B 0,C 180,E1 -9284.529,E2 -9284.529} C_VEL
LIN {X 0,Y 432.426,Z 323.502,A -85,B 0,C 180,E1 -9284.59,E2 -9284.59} C_VEL
LIN {X 0,Y 432.926,Z 311.657,A -85,B 0,C 180,E1 -9287.477,E2 -9287.477} C_VEL
LIN {X 0,Y 433.465,Z 299.943,A -85,B 0,C 180,E1 -9290.401,E2 -9290.401} C_VEL
LIN {X 0,Y 432.679,Z 293.05,A -85,B 0,C 180,E1 -9292.203,E2 -9292.203} C_VEL
LIN {X 0,Y 432.412,Z 291.548,A -85,B 0,C 180,E1 -9292.631,E2 -9292.631} C_VEL
LIN {X 0,Y 432.316,Z 291.445,A -85,B 0,C 180,E1 -9296.035,E2 -9296.035} C_VEL
LIN {X 0,Y 432.324,Z 291.444,A -85,B 0,C 180,E1 -9299.188,E2 -9299.188} C_VEL
LIN {X 0,Y 432.319,Z 291.442,A -85,B 0,C 180,E1 -9302.442,E2 -9302.442} C_VEL
LIN {X 0,Y 432.333,Z 291.443,A -85,B 0,C 180,E1 -9305.817,E2 -9305.817} C_VEL
LIN {X 0,Y 432.298,Z 291.451,A -85,B 0,C 180,E1 -9309.347,E2 -9309.347} C_VEL
LIN {X 0,Y 432.298,Z 291.446,A -85,B 0,C 180,E1 -9311.8,E2 -9311.8} C_VEL
LIN {X 0,Y 432.328,Z 291.441,A -85,B 0,C 180,E1 -9314.347,E2 -9314.347} C_VEL
LIN {X 0,Y 432.296,Z 291.451,A -85,B 0,C 180,E1 -9317.018,E2 -9317.018} C_VEL
LIN {X 0,Y 432.302,Z 291.444,A -85,B 0,C 180,E1 -9319.824,E2 -9319.824} C_VEL
LIN {X 0,Y 432.297,Z 291.451,A -85,B 0,C 180,E1 -9323.021,E2 -9323.021} C_VEL
LIN {X 0,Y 432.325,Z 291.441,A -85,B 0,C 180,E1 -9326.001,E2 -9326.001} C_VEL
LIN {X 0,Y 432.333,Z 291.441,A -85,B 0,C 180,E1 -9329.491,E2 -9329.491} C_VEL
LIN {X 0,Y 432.311,Z 291.443,A -85,B 0,C 180,E1 -9331.872,E2 -9331.872} C_VEL
LIN {X 0,Y 432.313,Z 291.446,A -85,B 0,C 180,E1 -9334.996,E2 -9334.996} C_VEL
LIN {X 0,Y 432.346,Z 291.44,A -85,B 0,C 180,E1 -9338.045,E2 -9338.045} C_VEL
LIN {X 0,Y 432.371,Z 291.437,A -85,B 0,C 180,E1 -9341.029,E2 -9341.029} C_VEL
LIN {X 0,Y 432.375,Z 291.437,A -85,B 0,C 180,E1 -9343.959,E2 -9343.959} C_VEL
LIN {X 0,Y 432.449,Z 291.427,A -85,B 0,C 180,E1 -9347.803,E2 -9347.803} C_VEL
LIN {X 0,Y 432.453,Z 291.426,A -85,B 0,C 180,E1 -9351.589,E2 -9351.589} C_VEL
LIN {X 0,Y 432.561,Z 291.416,A -85,B 0,C 180,E1 -9354.406,E2 -9354.406} C_VEL
LIN {X 0,Y 432.584,Z 291.416,A -85,B 0,C 180,E1 -9358.138,E2 -9358.138} C_VEL
LIN {X 0,Y 432.609,Z 291.413,A -85,B 0,C 180,E1 -9360,E2 -9360} C_VEL
LIN {X 0,Y 432.545,Z 291.414,A -85,B 0,C 180,E1 -9362.794,E2 -9362.794} C_VEL
LIN {X 0,Y 432.56,Z 291.416,A -85,B 0,C 180,E1 -9365.594,E2 -9365.594} C_VEL
LIN {X 0,Y 432.435,Z 291.429,A -85,B 0,C 180,E1 -9368.411,E2 -9368.411} C_VEL
LIN {X 0,Y 432.443,Z 291.428,A -85,B 0,C 180,E1 -9372.197,E2 -9372.197} C_VEL
LIN {X 0,Y 432.378,Z 291.437,A -85,B 0,C 180,E1 -9376.041,E2 -9376.041} C_VEL
LIN {X 0,Y 432.376,Z 291.442,A -85,B 0,C 180,E1 -9379.485,E2 -9379.485} C_VEL
LIN {X 0,Y 432.294,Z 291.447,A -85,B 0,C 180,E1 -9382.966,E2 -9382.966} C_VEL
LIN {X 0,Y 432.308,Z 291.444,A -85,B 0,C 180,E1 -9386.036,E2 -9386.036} C_VEL
LIN {X 0,Y 432.313,Z 291.449,A -85,B 0,C 180,E1 -9389.19,E2 -9389.19} C_VEL
LIN {X 0,Y 432.311,Z 291.443,A -85,B 0,C 180,E1 -9392.444,E2 -9392.444} C_VEL
LIN {X 0,Y 432.328,Z 291.441,A -85,B 0,C 180,E1 -9395.819,E2 -9395.819} C_VEL
LIN {X 0,Y 432.294,Z 291.449,A -85,B 0,C 180,E1 -9399.349,E2 -9399.349} C_VEL
LIN {X 0,Y 432.296,Z 291.445,A -85,B 0,C 180,E1 -9401.801,E2 -9401.801} C_VEL
LIN {X 0,Y 432.327,Z 291.442,A -85,B 0,C 180,E1 -9404.348,E2 -9404.348} C_VEL
LIN {X 0,Y 432.296,Z 291.45,A -85,B 0,C 180,E1 -9407.019,E2 -9407.019} C_VEL
LIN {X 0,Y 432.283,Z 291.446,A -85,B 0,C 180,E1 -9409.829,E2 -9409.829} C_VEL
LIN {X 0,Y 432.297,Z 291.448,A -85,B 0,C 180,E1 -9413.022,E2 -9413.022} C_VEL
LIN {X 0,Y 432.328,Z 291.442,A -85,B 0,C 180,E1 -9416.003,E2 -9416.003} C_VEL
LIN {X 0,Y 432.337,Z 291.439,A -85,B 0,C 180,E1 -9419.492,E2 -9419.492} C_VEL
LIN {X 0,Y 432.316,Z 291.443,A -85,B 0,C 180,E1 -9421.873,E2 -9421.873} C_VEL
LIN {X 0,Y 432.321,Z 291.446,A -85,B 0,C 180,E1 -9424.998,E2 -9424.998} C_VEL
LIN {X 0,Y 432.431,Z 291.59,A -85,B 0,C 180,E1 -9427.433,E2 -9427.433} C_VEL
LIN {X 0,Y 433.372,Z 297.815,A -85,B 0,C 180,E1 -9429.098,E2 -9429.098} C_VEL
LIN {X 0,Y 433.363,Z 303.729,A -85,B 0,C 180,E1 -9430.597,E2 -9430.597} C_VEL
LIN {X 0,Y 432.684,Z 317.333,A -85,B 0,C 180,E1 -9433.971,E2 -9433.971} C_VEL
LIN {X 0,Y 432.414,Z 323.595,A -85,B 0,C 180,E1 -9435.47,E2 -9435.47} C_VEL
LIN {X 0,Y 432.777,Z 326.242,A -85,B 0,C 180,E1 -9435.585,E2 -9435.585} C_VEL
LIN {X 0,Y 435.124,Z 341.923,A -85,B 0,C 180,E1 -9435.926,E2 -9435.926} C_VEL
LIN {X 0,Y 434.685,Z 399.119,A -85,B 0,C 180,E1 -9436.885,E2 -9436.885} C_VEL
LIN {X 0,Y 434.429,Z 408.484,A -85,B 0,C 180,E1 -9437.148,E2 -9437.148} C_VEL
LIN {X 0,Y 434.184,Z 416.936,A -85,B 0,C 180,E1 -9437.497,E2 -9437.497} C_VEL
LIN {X 0,Y 433.809,Z 425.428,A -85,B 0,C 180,E1 -9437.961,E2 -9437.961} C_VEL
LIN {X 0,Y 433.49,Z 433.753,A -85,B 0,C 180,E1 -9438.545,E2 -9438.545} C_VEL
LIN {X 0,Y 433.063,Z 441.784,A -85,B 0,C 180,E1 -9439.244,E2 -9439.244} C_VEL
LIN {X 0,Y 432.639,Z 450.452,A -85,B 0,C 180,E1 -9440.179,E2 -9440.179} C_VEL
LIN {X 0,Y 432.135,Z 458.952,A -85,B 0,C 180,E1 -9441.348,E2 -9441.348} C_VEL
LIN {X 0,Y 431.819,Z 465.621,A -85,B 0,C 180,E1 -9442.519,E2 -9442.519} C_VEL
LIN {X 0,Y 431.629,Z 469.998,A -85,B 0,C 180,E1 -9443.455,E2 -9443.455} C_VEL
LIN {X 0,Y 431.423,Z 475.156,A -85,B 0,C 180,E1 -9444.86,E2 -9444.86} C_VEL
LIN {X 0,Y 431.25,Z 478.943,A -85,B 0,C 180,E1 -9446.262,E2 -9446.262} C_VEL
LIN {X 0,Y 431.252,Z 480.683,A -85,B 0,C 180,E1 -9447.198,E2 -9447.198} C_VEL
LIN {X 0,Y 431.203,Z 481.93,A -85,B 0,C 180,E1 -9448.132,E2 -9448.132} C_VEL
LIN {X 0,Y 431.146,Z 482.706,A -85,B 0,C 180,E1 -9449.066,E2 -9449.066} C_VEL
LIN {X 0,Y 431.119,Z 483,A -85,B 0,C 180,E1 -9450,E2 -9450} C_VEL
LIN {X 0,Y 431.146,Z 482.705,A -85,B 0,C 180,E1 -9450.934,E2 -9450.934} C_VEL
LIN {X 0,Y 431.203,Z 481.925,A -85,B 0,C 180,E1 -9451.868,E2 -9451.868} C_VEL
LIN {X 0,Y 431.252,Z 480.675,A -85,B 0,C 180,E1 -9452.802,E2 -9452.802} C_VEL
LIN {X 0,Y 431.278,Z 477.781,A -85,B 0,C 180,E1 -9454.205,E2 -9454.205} C_VEL
LIN {X 0,Y 431.423,Z 475.143,A -85,B 0,C 180,E1 -9455.14,E2 -9455.14} C_VEL
LIN {X 0,Y 431.629,Z 469.977,A -85,B 0,C 180,E1 -9456.545,E2 -9456.545} C_VEL
LIN {X 0,Y 431.911,Z 463.17,A -85,B 0,C 180,E1 -9457.95,E2 -9457.95} C_VEL
LIN {X 0,Y 432.302,Z 455.724,A -85,B 0,C 180,E1 -9459.12,E2 -9459.12} C_VEL
LIN {X 0,Y 432.714,Z 448.379,A -85,B 0,C 180,E1 -9460.055,E2 -9460.055} C_VEL
LIN {X 0,Y 433.143,Z 440.511,A -85,B 0,C 180,E1 -9460.872,E2 -9460.872} C_VEL
LIN {X 0,Y 433.575,Z 432.195,A -85,B 0,C 180,E1 -9461.571,E2 -9461.571} C_VEL
LIN {X 0,Y 434.016,Z 421.574,A -85,B 0,C 180,E1 -9462.27,E2 -9462.27} C_VEL
LIN {X 0,Y 434.373,Z 410.018,A -85,B 0,C 180,E1 -9462.794,E2 -9462.794} C_VEL
LIN {X 0,Y 434.622,Z 400.347,A -85,B 0,C 180,E1 -9463.084,E2 -9463.084} C_VEL
LIN {X 0,Y 434.925,Z 339.772,A -85,B 0,C 180,E1 -9464.112,E2 -9464.112} C_VEL
LIN {X 0,Y 432.444,Z 324.044,A -85,B 0,C 180,E1 -9464.481,E2 -9464.481} C_VEL
LIN {X 0,Y 432.437,Z 322.289,A -85,B 0,C 180,E1 -9464.807,E2 -9464.807} C_VEL
LIN {X 0,Y 433.018,Z 309.502,A -85,B 0,C 180,E1 -9467.961,E2 -9467.961} C_VEL
LIN {X 0,Y 433.454,Z 299.742,A -85,B 0,C 180,E1 -9470.401,E2 -9470.401} C_VEL
LIN {X 0,Y 432.802,Z 293.884,A -85,B 0,C 180,E1 -9471.93,E2 -9471.93} C_VEL
LIN {X 0,Y 432.409,Z 291.508,A -85,B 0,C 180,E1 -9472.624,E2 -9472.624} C_VEL
LIN {X 0,Y 432.315,Z 291.445,A -85,B 0,C 180,E1 -9476.035,E2 -9476.035} C_VEL
LIN {X 0,Y 432.322,Z 291.445,A -85,B 0,C 180,E1 -9479.188,E2 -9479.188} C_VEL
LIN {X 0,Y 432.317,Z 291.442,A -85,B 0,C 180,E1 -9482.443,E2 -9482.443} C_VEL
LIN {X 0,Y 432.331,Z 291.442,A -85,B 0,C 180,E1 -9485.817,E2 -9485.817} C_VEL
LIN {X 0,Y 432.297,Z 291.451,A -85,B 0,C 180,E1 -9489.347,E2 -9489.347} C_VEL
LIN {X 0,Y 432.297,Z 291.446,A -85,B 0,C 180,E1 -9491.8,E2 -9491.8} C_VEL
LIN {X 0,Y 432.327,Z 291.441,A -85,B 0,C 180,E1 -9494.347,E2 -9494.347} C_VEL
LIN {X 0,Y 432.295,Z 291.452,A -85,B 0,C 180,E1 -9497.018,E2 -9497.018} C_VEL
LIN {X 0,Y 432.282,Z 291.447,A -85,B 0,C 180,E1 -9499.827,E2 -9499.827} C_VEL
LIN {X 0,Y 432.296,Z 291.451,A -85,B 0,C 180,E1 -9503.021,E2 -9503.021} C_VEL
LIN {X 0,Y 432.324,Z 291.441,A -85,B 0,C 180,E1 -9506.001,E2 -9506.001} C_VEL
LIN {X 0,Y 432.332,Z 291.441,A -85,B 0,C 180,E1 -9509.491,E2 -9509.491} C_VEL
LIN {X 0,Y 432.31,Z 291.443,A -85,B 0,C 180,E1 -9511.872,E2 -9511.872} C_VEL
LIN {X 0,Y 432.313,Z 291.446,A -85,B 0,C 180,E1 -9514.997,E2 -9514.997} C_VEL
LIN {X 0,Y 432.345,Z 291.44,A -85,B 0,C 180,E1 -9518.045,E2 -9518.045} C_VEL
LIN {X 0,Y 432.37,Z 291.437,A -85,B 0,C 180,E1 -9521.029,E2 -9521.029} C_VEL
LIN {X 0,Y 432.375,Z 291.437,A -85,B 0,C 180,E1 -9523.959,E2 -9523.959} C_VEL
LIN {X 0,Y 432.449,Z 291.427,A -85,B 0,C 180,E1 -9527.803,E2 -9527.803} C_VEL
LIN {X 0,Y 432.451,Z 291.426,A -85,B 0,C 180,E1 -9531.59,E2 -9531.59} C_VEL
LIN {X 0,Y 432.56,Z 291.416,A -85,B 0,C 180,E1 -9534.406,E2 -9534.406} C_VEL
LIN {X 0,Y 432.584,Z 291.416,A -85,B 0,C 180,E1 -9538.138,E2 -9538.138} C_VEL
LIN {X 0,Y 432.609,Z 291.413,A -85,B 0,C 180,E1 -9540,E2 -9540} C_VEL
LIN {X 0,Y 432.545,Z 291.414,A -85,B 0,C 180,E1 -9542.794,E2 -9542.794} C_VEL
LIN {X 0,Y 432.56,Z 291.416,A -85,B 0,C 180,E1 -9545.594,E2 -9545.594} C_VEL
LIN {X 0,Y 432.435,Z 291.429,A -85,B 0,C 180,E1 -9548.411,E2 -9548.411} C_VEL
LIN {X 0,Y 432.444,Z 291.428,A -85,B 0,C 180,E1 -9552.197,E2 -9552.197} C_VEL
LIN {X 0,Y 432.375,Z 291.438,A -85,B 0,C 180,E1 -9556.041,E2 -9556.041} C_VEL
LIN {X 0,Y 432.377,Z 291.441,A -85,B 0,C 180,E1 -9559.485,E2 -9559.485} C_VEL
LIN {X 0,Y 432.294,Z 291.447,A -85,B 0,C 180,E1 -9562.966,E2 -9562.966} C_VEL
LIN {X 0,Y 432.308,Z 291.444,A -85,B 0,C 180,E1 -9566.036,E2 -9566.036} C_VEL
LIN {X 0,Y 432.312,Z 291.449,A -85,B 0,C 180,E1 -9569.19,E2 -9569.19} C_VEL
LIN {X 0,Y 432.308,Z 291.444,A -85,B 0,C 180,E1 -9572.444,E2 -9572.444} C_VEL
LIN {X 0,Y 432.328,Z 291.441,A -85,B 0,C 180,E1 -9575.819,E2 -9575.819} C_VEL
LIN {X 0,Y 432.294,Z 291.449,A -85,B 0,C 180,E1 -9579.349,E2 -9579.349} C_VEL
LIN {X 0,Y 432.297,Z 291.445,A -85,B 0,C 180,E1 -9581.802,E2 -9581.802} C_VEL
LIN {X 0,Y 432.328,Z 291.442,A -85,B 0,C 180,E1 -9584.348,E2 -9584.348} C_VEL
LIN {X 0,Y 432.297,Z 291.45,A -85,B 0,C 180,E1 -9587.019,E2 -9587.019} C_VEL
LIN {X 0,Y 432.284,Z 291.446,A -85,B 0,C 180,E1 -9589.829,E2 -9589.829} C_VEL
LIN {X 0,Y 432.298,Z 291.448,A -85,B 0,C 180,E1 -9593.022,E2 -9593.022} C_VEL
LIN {X 0,Y 432.329,Z 291.441,A -85,B 0,C 180,E1 -9596.003,E2 -9596.003} C_VEL
LIN {X 0,Y 432.329,Z 291.441,A -85,B 0,C 180,E1 -9599.494,E2 -9599.494} C_VEL
LIN {X 0,Y 432.312,Z 291.444,A -85,B 0,C 180,E1 -9601.873,E2 -9601.873} C_VEL
LIN {X 0,Y 432.321,Z 291.447,A -85,B 0,C 180,E1 -9604.998,E2 -9604.998} C_VEL
LIN {X 0,Y 432.414,Z 291.614,A -85,B 0,C 180,E1 -9607.492,E2 -9607.492} C_VEL
LIN {X 0,Y 433.316,Z 297.614,A -85,B 0,C 180,E1 -9609.095,E2 -9609.095} C_VEL
LIN {X 0,Y 433.364,Z 303.528,A -85,B 0,C 180,E1 -9610.598,E2 -9610.598} C_VEL
LIN {X 0,Y 432.686,Z 317.13,A -85,B 0,C 180,E1 -9613.971,E2 -9613.971} C_VEL
LIN {X 0,Y 432.412,Z 323.76,A -85,B 0,C 180,E1 -9615.538,E2 -9615.538} C_VEL
LIN {X 0,Y 433.207,Z 328.9,A -85,B 0,C 180,E1 -9615.694,E2 -9615.694} C_VEL
LIN {X 0,Y 435.022,Z 340.53,A -85,B 0,C 180,E1 -9615.949,E2 -9615.949} C_VEL
LIN {X 0,Y 434.698,Z 399.681,A -85,B 0,C 180,E1 -9616.948,E2 -9616.948} C_VEL
LIN {X 0,Y 434.427,Z 408.758,A -85,B 0,C 180,E1 -9617.207,E2 -9617.207} C_VEL
LIN {X 0,Y 434.116,Z 418.346,A -85,B 0,C 180,E1 -9617.614,E2 -9617.614} C_VEL
LIN {X 0,Y 433.687,Z 428.391,A -85,B 0,C 180,E1 -9618.195,E2 -9618.195} C_VEL
LIN {X 0,Y 433.291,Z 438.431,A -85,B 0,C 180,E1 -9618.977,E2 -9618.977} C_VEL
LIN {X 0,Y 432.387,Z 443.363,A -85,B 0,C 180,E1 -9619.426,E2 -9619.426} C_VEL
LIN {X 0,Y 429.077,Z 450.817,A -85,B 0,C 180,E1 -9620.189,E2 -9620.189} C_VEL
LIN {X 0,Y 425.822,Z 457.585,A -85,B 0,C 180,E1 -9621.049,E2 -9621.049} C_VEL
LIN {X 0,Y 424.982,Z 461.255,A -85,B 0,C 180,E1 -9621.64,E2 -9621.64} C_VEL
LIN {X 0,Y 424.681,Z 467.719,A -85,B 0,C 180,E1 -9622.871,E2 -9622.871} C_VEL
LIN {X 0,Y 424.42,Z 473.481,A -85,B 0,C 180,E1 -9624.298,E2 -9624.298} C_VEL
LIN {X 0,Y 424.268,Z 476.49,A -85,B 0,C 180,E1 -9625.249,E2 -9625.249} C_VEL
LIN {X 0,Y 424.161,Z 478.822,A -85,B 0,C 180,E1 -9626.2,E2 -9626.2} C_VEL
LIN {X 0,Y 424.152,Z 480.598,A -85,B 0,C 180,E1 -9627.151,E2 -9627.151} C_VEL
LIN {X 0,Y 424.13,Z 481.879,A -85,B 0,C 180,E1 -9628.101,E2 -9628.101} C_VEL
LIN {X 0,Y 424.068,Z 482.689,A -85,B 0,C 180,E1 -9629.05,E2 -9629.05} C_VEL
LIN {X 0,Y 424.04,Z 482.998,A -85,B 0,C 180,E1 -9630,E2 -9630} C_VEL
LIN {X 0,Y 424.068,Z 482.721,A -85,B 0,C 180,E1 -9630.95,E2 -9630.95} C_VEL
LIN {X 0,Y 424.127,Z 481.976,A -85,B 0,C 180,E1 -9631.899,E2 -9631.899} C_VEL
LIN {X 0,Y 424.142,Z 480.76,A -85,B 0,C 180,E1 -9632.849,E2 -9632.849} C_VEL
LIN {X 0,Y 424.197,Z 477.901,A -85,B 0,C 180,E1 -9634.276,E2 -9634.276} C_VEL
LIN {X 0,Y 424.342,Z 475.301,A -85,B 0,C 180,E1 -9635.226,E2 -9635.226} C_VEL
LIN {X 0,Y 424.493,Z 471.521,A -85,B 0,C 180,E1 -9636.32,E2 -9636.32} C_VEL
LIN {X 0,Y 424.693,Z 467.132,A -85,B 0,C 180,E1 -9637.344,E2 -9637.344} C_VEL
LIN {X 0,Y 424.924,Z 462.058,A -85,B 0,C 180,E1 -9638.321,E2 -9638.321} C_VEL
LIN {X 0,Y 425.285,Z 456.076,A -85,B 0,C 180,E1 -9639.272,E2 -9639.272} C_VEL
LIN {X 0,Y 425.725,Z 448.796,A -85,B 0,C 180,E1 -9640.222,E2 -9640.222} C_VEL
LIN {X 0,Y 426.13,Z 441.018,A -85,B 0,C 180,E1 -9641.053,E2 -9641.053} C_VEL
LIN {X 0,Y 426.514,Z 434.317,A -85,B 0,C 180,E1 -9641.645,E2 -9641.645} C_VEL
LIN {X 0,Y 426.885,Z 426.131,A -85,B 0,C 180,E1 -9642.237,E2 -9642.237} C_VEL
LIN {X 0,Y 427.274,Z 417.843,A -85,B 0,C 180,E1 -9642.709,E2 -9642.709} C_VEL
LIN {X 0,Y 427.522,Z 408.899,A -85,B 0,C 180,E1 -9643.094,E2 -9643.094} C_VEL
LIN {X 0,Y 427.771,Z 399.578,A -85,B 0,C 180,E1 -9643.365,E2 -9643.365} C_VEL
LIN {X 0,Y 428.061,Z 340.638,A -85,B 0,C 180,E1 -9644.378,E2 -9644.378} C_VEL
LIN {X 0,Y 425.451,Z 324.139,A -85,B 0,C 180,E1 -9644.774,E2 -9644.774} C_VEL
LIN {X 0,Y 425.416,Z 323.5,A -85,B 0,C 180,E1 -9644.836,E2 -9644.836} C_VEL
LIN {X 0,Y 425.96,Z 311.655,A -85,B 0,C 180,E1 -9647.772,E2 -9647.772} C_VEL
LIN {X 0,Y 426.47,Z 301.893,A -85,B 0,C 180,E1 -9650.247,E2 -9650.247} C_VEL
LIN {X 0,Y 425.985,Z 296.036,A -85,B 0,C 180,E1 -9651.79,E2 -9651.79} C_VEL
LIN {X 0,Y 425.346,Z 292.381,A -85,B 0,C 180,E1 -9652.847,E2 -9652.847} C_VEL
LIN {X 0,Y 425.258,Z 292.329,A -85,B 0,C 180,E1 -9655.447,E2 -9655.447} C_VEL
LIN {X 0,Y 425.305,Z 292.316,A -85,B 0,C 180,E1 -9658.859,E2 -9658.859} C_VEL
LIN {X 0,Y 425.26,Z 292.323,A -85,B 0,C 180,E1 -9661.926,E2 -9661.926} C_VEL
LIN {X 0,Y 425.291,Z 292.324,A -85,B 0,C 180,E1 -9665.336,E2 -9665.336} C_VEL
LIN {X 0,Y 425.276,Z 292.322,A -85,B 0,C 180,E1 -9668.9,E2 -9668.9} C_VEL
LIN {X 0,Y 425.251,Z 292.324,A -85,B 0,C 180,E1 -9672.655,E2 -9672.655} C_VEL
LIN {X 0,Y 425.28,Z 292.324,A -85,B 0,C 180,E1 -9675.282,E2 -9675.282} C_VEL
LIN {X 0,Y 425.243,Z 292.326,A -85,B 0,C 180,E1 -9678.617,E2 -9678.617} C_VEL
LIN {X 0,Y 425.277,Z 292.325,A -85,B 0,C 180,E1 -9681.099,E2 -9681.099} C_VEL
LIN {X 0,Y 425.287,Z 292.322,A -85,B 0,C 180,E1 -9684.663,E2 -9684.663} C_VEL
LIN {X 0,Y 425.252,Z 292.323,A -85,B 0,C 180,E1 -9688.072,E2 -9688.072} C_VEL
LIN {X 0,Y 425.288,Z 292.319,A -85,B 0,C 180,E1 -9691.365,E2 -9691.365} C_VEL
LIN {X 0,Y 425.25,Z 292.328,A -85,B 0,C 180,E1 -9694.552,E2 -9694.552} C_VEL
LIN {X 0,Y 425.282,Z 292.319,A -85,B 0,C 180,E1 -9697.73,E2 -9697.73} C_VEL
LIN {X 0,Y 425.35,Z 292.315,A -85,B 0,C 180,E1 -9700.703,E2 -9700.703} C_VEL
LIN {X 0,Y 425.309,Z 292.316,A -85,B 0,C 180,E1 -9703.685,E2 -9703.685} C_VEL
LIN {X 0,Y 425.384,Z 292.306,A -85,B 0,C 180,E1 -9707.096,E2 -9707.096} C_VEL
